(* PLC project WMT, Росатом LocalPLC 1, author Коробейников Петр *)
(* stored: creationDateTime 2021-03-09T09:02:31, contentDescription Система предиктивной диагностики. Модель теплового режима., productRelease 1, modificationDateTime 2023-03-16T09:01:23, language ru-RU, version 1, organization Филиал ВНИИЭФ НИИИС *)

TYPE P_INT : STRUCT
  A : INT := -1;
  B : INT := -1;
END_STRUCT;
END_TYPE

TYPE P_UINT : STRUCT
  A : UINT := 0;
  B : UINT := 0;
END_STRUCT;
END_TYPE

TYPE P_SINT : STRUCT
  A : SINT;
  B : SINT;
END_STRUCT;
END_TYPE

TYPE P_IDPIT : STRUCT
  A : UINT := 0;
  B : TPos8 := -1;
END_STRUCT;
END_TYPE

TYPE P_SIBT : STRUCT
  A : SINT := 0;
  B : BYTE := 0;
END_STRUCT;
END_TYPE

TYPE P_BOOL : STRUCT
  A : BOOL := false;
  B : BOOL := false;
END_STRUCT;
END_TYPE

TYPE TDef : STRUCT
  ID : UINT := 0;
  CF : WORD := 0;
  R0 : INT := 0;
  XYZ : ARRAY[0..2] OF INT := [0, 0, 0];
  LWH : ARRAY[0..2] OF INT := [100, 100, 100];
  Ig : SINT := 0;
  Im : SINT := 0;
  Iv : SINT := 0;
END_STRUCT;
END_TYPE

TYPE TMat : STRUCT
  KT : REAL := 0.11;
  CP : REAL := 1666.0;
  PL : REAL := 880.3;
  MD : REAL := 198.1;
END_STRUCT;
END_TYPE

TYPE TRad : STRUCT
  Vm : REAL := 0.02;
  Fk : REAL := 1.1;
  Q0 : REAL := 0.003;
  Q1 : REAL := 0.01;
  BL : ARRAY[0..3] OF REAL := [0.2, 0.6, 0.85, 1.0];
END_STRUCT;
END_TYPE

TYPE THead : STRUCT
  Ni : SINT := 0;
  Ng : SINT := 0;
  Nm : SINT := 0;
  Nv : SINT := 0;
  Np : SINT := 0;
  Ri : SINT := 0;
  ID : UINT := 0;
  TR : ARRAY[0..3] OF TIME := [T#60s, T#30s, T#10s, T#5s];
  Ax : UINT := 0;
  pX : INT := 0;
  pY : INT := 0;
  pZ : INT := 0;
  RV : ARRAY[0..1] OF DINT := [0, 0];
END_STRUCT;
END_TYPE

TYPE TRes : STRUCT
  DR : UDINT := 0;
  TR : TIME := T#0s;
  FP : TIME := T#0s;
  ER : UINT := 0;
  FL : WORD := 0;
  RV : ARRAY[0..5] OF UDINT := [0, 0, 0, 0, 0, 0];
END_STRUCT;
END_TYPE

TYPE TVal : STRUCT
  Iv : INT := 0;
  Vi : ARRAY[0..2] OF P_SINT := [0, 0, 0];
END_STRUCT;
END_TYPE

TYPE TProf : ARRAY[0..11] OF P_SINT;
END_TYPE

TYPE TConf : STRUCT
  Nm : UINT := 0;
  Nr : UINT := 0;
  Tc : TIME := T#10s;
END_STRUCT;
END_TYPE

TYPE TPhaseI : STRUCT
  Ic : REAL := 100.0;
  Tin : REAL := 40.0;
  Tout : REAL := 80.0;
  Rn : DWORD := 16#FFFF;
  RD : ARRAY[0..7] OF P_SINT := [0, 0, 0, 0, 0, 0, 0, 0];
END_STRUCT;
END_TYPE

TYPE TPhaseO : STRUCT
  Q0 : REAL := 0.0;
  Q1 : REAL := 0.0;
  Q2 : REAL := 0.0;
  Tin : REAL := 20.0;
  Tout : REAL := 80.0;
  Qm : REAL := 0.01;
  Se : REAL := 0.01;
  Ve : REAL := 0.01;
END_STRUCT;
END_TYPE

TYPE TCond : STRUCT
  ID : UINT := 0;
  Tmid : INT := 0;
  Tmin : TDot;
  Tmax : TDot;
END_STRUCT;
END_TYPE

TYPE TVarI : STRUCT
  DTI : UDINT := 0;
  TMI : TIME := T#0s;
  TOV : REAL := 0.0;
  MHT : REAL := 0.0;
  RI1 : REAL := 0.0;
  RI2 : REAL := 0.0;
END_STRUCT;
END_TYPE

TYPE TVarO : STRUCT
  DTO : UDINT := 0;
  TMO : TIME := T#0s;
  QTY : REAL := 0.0;
  QTS : REAL := 0.0;
  RO1 : REAL := 0.0;
  RO2 : REAL := 0.0;
END_STRUCT;
END_TYPE

TYPE TError : (E_SUCCESS, E_ID, E_HEAD, E_INDEX, E_ITEMPOS, E_ITEM, E_GRID, E_AXIS, E_PRIO, E_MATER, E_PROFILE, E_VALUE, E_STACKSIZE, E_ROOT, E_ITEMSIZE, E_STEPSIZE, E_TIMESIZE, E_NOTREADY, E_STRUCT, E_VALIDATE, E_LOC2ABS, E_ABS2LOC, E_GETTEMP, E_SETTEMP, E_CHECKVALID, E_LINKITEMS, E_PROCESS, E_PREPROC, E_POSTPROC, E_BADTEMP, E_STATE, E_CHECK, E_FAIL, W_PERIOD) := E_SUCCESS;
END_TYPE

TYPE TDir : (DIR_UP, DIR_DOWN);
END_TYPE

TYPE TIter : STRUCT
  dir : TDir := DIR_UP;
  prev : TPos8 := -1;
  item : TPos8 := -1;
  next : TPos8 := -1;
  last : TPos8 := -1;
  stack : ARRAY[0..3] OF TPos8 := [0, 0, 0, 0];
END_STRUCT;
END_TYPE

TYPE TPoint : ARRAY[0..2] OF REAL;
END_TYPE

TYPE TAxO : STRUCT
  x : USINT := 0;
  y : USINT := 0;
  z : USINT := 0;
END_STRUCT;
END_TYPE

TYPE P_RESI : STRUCT
  A : REAL := 0.0;
  B : SINT := 0;
END_STRUCT;
END_TYPE

TYPE P_RERE : STRUCT
  A : REAL := 0.0;
  B : REAL := 0.0;
END_STRUCT;
END_TYPE

TYPE TMatter : STRUCT
  a : REAL := 0.0001;
  l : REAL := 1.0;
  h : REAL := 0.001;
  k : REAL := 1.0;
END_STRUCT;
END_TYPE

TYPE TProps : STRUCT
  Air : BOOL := false;
  Oil : BOOL := false;
  Fluid : BOOL := false;
  Solid : BOOL := false;
END_STRUCT;
END_TYPE

TYPE LOGLEVEL : (CRITICAL, WARNING, INFO, DEBUG) := DEBUG;
END_TYPE

TYPE TStat : STRUCT
  RDY : BOOL := FALSE;
  DBG : BOOL := TRUE;
  ERR : TError := E_SUCCESS;
  PAR : UINT := 0;
  STR : STRING := '';
END_STRUCT;
END_TYPE

TYPE TGrid : STRUCT
  A : ARRAY[0..6271] OF TVar;
END_STRUCT;
END_TYPE

TYPE TVar : DINT;
END_TYPE

TYPE TDot : STRUCT
  V : INT := 0;
  A : TKnot := [0, 0, 0];
END_STRUCT;
END_TYPE

TYPE TShape : STRUCT
  wF : WORD := 0;
  Kn : TKnot := [0, 0, 0];
  p0 : TPoint := [0.0, 0.0, 0.0];
  pL : TPoint := [0.0, 0.0, 0.0];
  Lx : TPoint := [0.0, 0.0, 0.0];
END_STRUCT;
END_TYPE

TYPE TKnot : ARRAY[0..2] OF INT := [0, 0, 0];
END_TYPE

TYPE TItem : STRUCT
  ID : UINT := 0;
  Im : SINT := -1;
  Iv : SINT := -1;
  PDT : ARRAY[0..2] OF DT := [t#0ms, t#0ms, t#0ms];
  Par : TPos8 := -1;
  Num : SINT := 0;
  Kids : ARRAY[0..15] OF TPos8 := [0, 0, 0, 0, 0, 0, 0, 0, 0, 0, 0, 0, 0, 0, 0, 0];
END_STRUCT;
END_TYPE

TYPE TPos16 : INT := -1;
END_TYPE

TYPE TPos8 : SINT := -1;
END_TYPE

TYPE TItems : STRUCT
  Pr : ARRAY[0..99] OF P_IDPIT := [0, 0, 0, 0, 0, 0, 0, 0, 0, 0, 0, 0, 0, 0, 0, 0, 0, 0, 0, 0, 0, 0, 0, 0, 0, 0, 0, 0, 0, 0, 0, 0, 0, 0, 0, 0, 0, 0, 0, 0, 0, 0, 0, 0, 0, 0, 0, 0, 0, 0, 0, 0, 0, 0, 0, 0, 0, 0, 0, 0, 0, 0, 0, 0, 0, 0, 0, 0, 0, 0, 0, 0, 0, 0, 0, 0, 0, 0, 0, 0, 0, 0, 0, 0, 0, 0, 0, 0, 0, 0, 0, 0, 0, 0, 0, 0, 0, 0, 0, 0];
  It : ARRAY[0..99] OF TItem := [0, 0, 0, 0, 0, 0, 0, 0, 0, 0, 0, 0, 0, 0, 0, 0, 0, 0, 0, 0, 0, 0, 0, 0, 0, 0, 0, 0, 0, 0, 0, 0, 0, 0, 0, 0, 0, 0, 0, 0, 0, 0, 0, 0, 0, 0, 0, 0, 0, 0, 0, 0, 0, 0, 0, 0, 0, 0, 0, 0, 0, 0, 0, 0, 0, 0, 0, 0, 0, 0, 0, 0, 0, 0, 0, 0, 0, 0, 0, 0, 0, 0, 0, 0, 0, 0, 0, 0, 0, 0, 0, 0, 0, 0, 0, 0, 0, 0, 0, 0];
  Sh : ARRAY[0..100] OF TShape := [0, 0, 0, 0, 0, 0, 0, 0, 0, 0, 0, 0, 0, 0, 0, 0, 0, 0, 0, 0, 0, 0, 0, 0, 0, 0, 0, 0, 0, 0, 0, 0, 0, 0, 0, 0, 0, 0, 0, 0, 0, 0, 0, 0, 0, 0, 0, 0, 0, 0, 0, 0, 0, 0, 0, 0, 0, 0, 0, 0, 0, 0, 0, 0, 0, 0, 0, 0, 0, 0, 0, 0, 0, 0, 0, 0, 0, 0, 0, 0, 0, 0, 0, 0, 0, 0, 0, 0, 0, 0, 0, 0, 0, 0, 0, 0, 0, 0, 0, 0, 0];
  Cn : ARRAY[0..100] OF TCond := [0, 0, 0, 0, 0, 0, 0, 0, 0, 0, 0, 0, 0, 0, 0, 0, 0, 0, 0, 0, 0, 0, 0, 0, 0, 0, 0, 0, 0, 0, 0, 0, 0, 0, 0, 0, 0, 0, 0, 0, 0, 0, 0, 0, 0, 0, 0, 0, 0, 0, 0, 0, 0, 0, 0, 0, 0, 0, 0, 0, 0, 0, 0, 0, 0, 0, 0, 0, 0, 0, 0, 0, 0, 0, 0, 0, 0, 0, 0, 0, 0, 0, 0, 0, 0, 0, 0, 0, 0, 0, 0, 0, 0, 0, 0, 0, 0, 0, 0, 0, 0];
  Gr : ARRAY[0..99] OF TGrid := [0, 0, 0, 0, 0, 0, 0, 0, 0, 0, 0, 0, 0, 0, 0, 0, 0, 0, 0, 0, 0, 0, 0, 0, 0, 0, 0, 0, 0, 0, 0, 0, 0, 0, 0, 0, 0, 0, 0, 0, 0, 0, 0, 0, 0, 0, 0, 0, 0, 0, 0, 0, 0, 0, 0, 0, 0, 0, 0, 0, 0, 0, 0, 0, 0, 0, 0, 0, 0, 0, 0, 0, 0, 0, 0, 0, 0, 0, 0, 0, 0, 0, 0, 0, 0, 0, 0, 0, 0, 0, 0, 0, 0, 0, 0, 0, 0, 0, 0, 0];
  Gr2 : ARRAY[0..1] OF TGrid2 := [0, 0];
END_STRUCT;
END_TYPE

TYPE TSets : STRUCT
  Mt : ARRAY[0..11] OF TMat := [0, 0, 0, 0, 0, 0, 0, 0, 0, 0, 0, 0];
  Vl : ARRAY[0..24] OF TVal := [0, 0, 0, 0, 0, 0, 0, 0, 0, 0, 0, 0, 0, 0, 0, 0, 0, 0, 0, 0, 0, 0, 0, 0, 0];
  Pr : ARRAY[0..29] OF TProf := [0, 0, 0, 0, 0, 0, 0, 0, 0, 0, 0, 0, 0, 0, 0, 0, 0, 0, 0, 0, 0, 0, 0, 0, 0, 0, 0, 0, 0, 0];
  Bf : ARRAY[0..31] OF REAL := [0, 0, 0, 0, 0, 0, 0, 0, 0, 0, 0, 0, 0, 0, 0, 0, 0, 0, 0, 0, 0, 0, 0, 0, 0, 0, 0, 0, 0, 0, 0, 0];
END_STRUCT;
END_TYPE

TYPE THandle : ULINT;
END_TYPE

TYPE TGrid2 : STRUCT
  A : ARRAY[0..12543] OF TVar;
END_STRUCT;
END_TYPE

(* Дескриптор массива ITS.GR *)
FUNCTION its_gr2 : THandle
  VAR_INPUT
    Off : TPos8 := 0;  (* Опорная позиция сетки *)
  END_VAR

            {{ ITS_GR2 = (THANDLE)&__GET_GLOBAL_ITS()->GR2.table[OFF]; }}

          
END_FUNCTION

(* Дескриптор массива ITS.GR *)
FUNCTION its_gr : THandle
  VAR_INPUT
    Off : TPos8 := 0;  (* Опорная позиция сетки *)
  END_VAR

            {{ ITS_GR = (THANDLE)&__GET_GLOBAL_ITS()->GR.table[OFF]; }}

          
END_FUNCTION

(* Возвращает фигуру элемента *)
FUNCTION get_sh : TShape
  VAR_INPUT
    PSH : TPos8 := -1;  (* Позиция фигуры элемента *)
  END_VAR

            {{ return (GET_SH = __GET_GLOBAL_ITS()->SH.table[PSH]); }}

          
END_FUNCTION

(* Поиск в массиве IDS по ID *)
FUNCTION ID2PIT : TPos8
  VAR_INPUT
    ID : UINT := 0;  (* Идентификатор элемента *)
  END_VAR
  VAR
    bFound : BOOL := false;  (* Флаг - элемент найден *)
  END_VAR

            {{
  ID2PIT = -1;
  P_IDPIT *IDS = &(__GET_GLOBAL_ITS()->PR.table[0]);
  if (ID != 0) {
    int lBound=0, rBound=99, test;
    if (IDS[rBound].A == ID)      ID2PIT = IDS[rBound].B;
    else if (IDS[lBound].A == ID) ID2PIT = IDS[lBound].B;
    else {
      if ( (IDS[lBound].A < ID) && (ID < IDS[rBound].A) ) {
        while (TRUE) {
          test = (lBound+rBound)/2;
          if (IDS[test].A == ID) { ID2PIT = IDS[test].B; break; }
          if (rBound-lBound <= 1) break;
          if (IDS[test].A <  ID) lBound = test; else rBound = test; 
        }
      }
    }
  } else ID2PIT = IDS[0].B;
}}
          
END_FUNCTION

(* TRUE, если элемент - родитель *)
FUNCTION is_poly : BOOL
  VAR_INPUT
    PIT : TPos8 := -1;  (* Позиция элемента *)
  END_VAR

            {{ 
  return (IS_POLY = (__GET_GLOBAL_ITS()->IT.table[PIT].NUM > 0)); 
}}

          
END_FUNCTION

(* Терминальный итератор *)
FUNCTION it_end : TIter
  VAR_INPUT
    PIT : TPos8 := -1;  (* Признак терминального узла *)
  END_VAR

            {{ 
  return (IT_END = ((TITER){ TDIR__DIR_UP, -1, -1, -1, -1, {0,0,0,0} } )); 
}}

          
END_FUNCTION

(* Аварийное завершение программы *)
FUNCTION halt : BOOL
  VAR_INPUT
    ERR : TError := E_FAIL;  (* Код ошибки *)
  END_VAR

            (* Использует вызов sleep() и exit() для завершения потоков *)
{{
  //#ifndef __ASSERT_H
  //#define __ASSERT_H 1
     //#include <unistd.h> // Include "unistd.h" for sleep() & exit() function
  //#endif // __ASSERT_H
  //sleep(3); // Wait for message logging..
  //exit(ERR);
}}
          
END_FUNCTION

(* Приоритет по коду ошибки *)
FUNCTION Err2Lev : LOGLEVEL
  VAR_INPUT
    Err : TError := E_SUCCESS;  (* Флаг ошибки *)
  END_VAR

            CASE Err OF
E_SUCCESS:  
  Err2Lev:=INFO;  
W_PERIOD:   
  Err2Lev:=WARNING;  
ELSE        
  Err2Lev:=CRITICAL;  
END_CASE;
RETURN;
          
END_FUNCTION

(* Выдает строку по коду ошибки *)
FUNCTION Err2Str : STRING
  VAR_INPUT
    ERR : TError := E_SUCCESS;  (* Код ошибки *)
  END_VAR

            case ERR of
(* Информационные сообщения *)
E_SUCCESS:      Err2Str := 'Succeeded!';

(* Критические ошибки *)
E_FAIL:         Err2Str := 'Unexpected error';
E_STATE:        Err2Str := 'Program state error';
E_CHECK:        Err2Str := 'Check point error';
E_HEAD:         Err2Str := 'Invalid head';
E_INDEX:        Err2Str := 'Invalid index';
E_ITEMPOS:      Err2Str := 'Invalid item position';
E_ITEM:         Err2Str := 'Invalid element';
E_GRID:         Err2Str := 'Invalid grid';
E_AXIS:         Err2Str := 'Invalid axis';
E_PRIO:         Err2Str := 'Invalid prio';
E_MATER:        Err2Str := 'Invalid mater';
E_PROFILE:      Err2Str := 'Invalid profile';
E_VALUE:        Err2Str := 'Invalid value';
E_ROOT:         Err2Str := 'Invalid ROOT';
E_ITEMSIZE:     Err2Str := 'Bad ItemAt size';
E_STEPSIZE:     Err2Str := 'Bad axis step';
E_TIMESIZE:     Err2Str := 'Bad time step';
E_STACKSIZE:    Err2Str := 'Small stacksize';
E_NOTREADY:     Err2Str := 'Object dont ready';
E_LOC2ABS:      Err2Str := 'Loc2Abs error';
E_ABS2LOC:      Err2Str := 'Abs2Loc error';
E_VALIDATE:     Err2Str := 'Validate error';
E_CHECKVALID:   Err2Str := 'CheckValid error';
E_LINKITEMS:    Err2Str := 'LinkItems error';
E_PROCESS:      Err2Str := 'Process item error';
E_BADTEMP:      Err2Str := 'GetTemp error';

(* Предупреждения *)
W_PERIOD:       Err2Str := 'Small period';
else            Err2Str := 'Unknown error';
end_case;

          
END_FUNCTION

(* Протоколирование ошибки *)
FUNCTION LogMsg : STRING
  VAR_INPUT
    STR : STRING := '';  (* Строка для протокола *)
    LVL : LOGLEVEL := DEBUG;  (* Уровень сообщения (по умолчанию - Debug) *)
    ERR : TError := E_SUCCESS;  (* Код ошибки *)
  END_VAR

            {{
  #ifdef _BEREMIZ_H_
    #define __LOG_MSG(level,string,length) LogMessage(level,(char *)string,length)
  #else
    #define __LOG_MSG(level,string,length) printf("%s\n", (char *)string)
  #endif
  TSTAT *pStat = __GET_GLOBAL_STAT();
  if (LVL!=LOGLEVEL__DEBUG || (LVL==LOGLEVEL__DEBUG && pStat->DBG)) {
    if (STR.len) __LOG_MSG(LVL, (char *)STR.body, STR.len);
  }
  if (ERR!=TERROR__E_SUCCESS) {
    pStat->ERR=ERR;
    LVL=ERR2LEV(1,NULL,ERR); 
    STR=ERR2STR(1,NULL,ERR);
    if (STR.len) __LOG_MSG(LVL,(char *)STR.body,STR.len);
  }
  return (LOGMSG = __INIT_STRING);
}}

          
END_FUNCTION

(* Выдает строку по коду ошибки *)
FUNCTION MakeMsg : STRING
  VAR_INPUT
    S0 : STRING := '';  (* Строка 0 *)
    S1 : STRING := '';  (* Строка 1 *)
    S2 : STRING := '';  (* Строка 2 *)
    S3 : STRING := '';  (* Строка 3 *)
  END_VAR
  VAR
    BLOG : BOOL := FALSE;  (* Флаг работы *)
  END_VAR

            {{ BLOG = __GET_GLOBAL_STAT()->DBG; }}
if (BLOG) then 
  MakeMsg:=concat(concat(concat(S0, S1), S2), S3); 
else 
  MakeMsg:=''; 
end_if;
          
END_FUNCTION

(* Аналог функции assert в C *)
FUNCTION assert : BOOL
  VAR_INPUT
    STAT : BOOL := FALSE;  (* Выражение для утверждения *)
    ERR : TError := E_FAIL;  (* Код ошибки *)
    STR : STRING := '';  (* Строка в лог *)
  END_VAR

            {{
//  #ifndef __ASSERT_H
//  #define __ASSERT_H 1
//     #include <unistd.h> // Include "unistd.h" for sleep() & exit() function
//     #include <assert.h> // Include "unistd.h" for sleep() & exit() function
//  #endif // __ASSERT_H
  if (!(ASSERT=STAT)) { 
    STR = MAKEMSG(1, NULL, 
      __STRING_LITERAL(27,"OpenPLC: ASSERTION FAILED! "), 
      STR,
      __INIT_STRING,
      __INIT_STRING
    );
    LOGMSG(1, NULL, STR, LOGLEVEL__CRITICAL, ERR); 
    //HALT(1, NULL, ERR);
    //sleep(3); // Wait for message logging..
    //exit(ERR);
//    assert(0);
  }
}}
          
END_FUNCTION

(* Уровень вложенности элемента *)
FUNCTION it_lev : SINT
  VAR_INPUT
    PIT : TPos8 := -1;
  END_VAR
  VAR
    IID : UINT := 16#ffff;
  END_VAR

            {{
  IID = __GET_GLOBAL_ITS()->IT.table[PIT].ID;
  if (IID==0 || IID==0xffff) return (IT_LEV=-1);
  IT_LEV = 3;
  if (IID & 0x000F) return(IT_LEV); IT_LEV--;
  if (IID & 0x00F0) return(IT_LEV); IT_LEV--;
  if (IID & 0x0F00) return(IT_LEV); IT_LEV--;
}}

          
END_FUNCTION

(* Обход дерева элементов *)
FUNCTION it_next : TIter
  VAR_INPUT
    it : TIter;  (* Итератор *)
  END_VAR

            {{ 
  /* Алгоритм обхода:
    1) Если предыдущий узел - родительский для этого узла 
       -> переходим к первому дочернему узлу (если нет->к родителю);
    2) Если предыдущий узел - дочерний для этого узла  
       -> переходим к следующему дочернему узлу (если нет->к родителю) 
  */
  SINT iSub = 0;
  SINT iLevel = 0;
  BOOL bBreak = FALSE;
  TITEM *Items = &(__GET_GLOBAL_ITS()->IT.table[0]);
  
  while (!bBreak && IT.ITEM!=(-1)) { 
    IT.ITEM = IT.NEXT;  // Переход к следующему элементу
    if (IT.ITEM!=(-1)) {
      // Запоминаем уровень текущего узла в стеке со смещением +1
      iLevel = IT_LEV(1,NULL,IT.ITEM)+1; 
      
      // Определение следующего узла
      if (IT.PREV == Items[IT.ITEM].PAR) {
        // предыдущий узел является является родительским узлом этого узла ->
        iSub = 0;
        if (Items[IT.ITEM].NUM > iSub) { 
          // ВНИЗ -> к первому дочернему узлу (если есть)
          IT.NEXT = Items[IT.ITEM].KIDS.table[iSub];
          IT.STACK.table[iLevel] = iSub;
          IT.DIR = TDIR__DIR_DOWN;  // Актуально если есть потомки
          bBreak = TRUE; 
        } else {    
          // ВВЕРХ -> к родителю (потомков нет)
          IT.NEXT = (IT.ITEM != IT.LAST) ? IT.NEXT = Items[IT.ITEM].PAR : (-1);
          IT.DIR = TDIR__DIR_UP;    // Актуально для любого элемента
          bBreak = TRUE;
        }
      } else if (Items[IT.PREV].PAR == IT.ITEM) { 
        // предыдущий узел является дочерним узлом этого узла ->
        iSub = IT.STACK.table[iLevel]+1;
        if (iSub < Items[IT.ITEM].NUM) {
          // ПО ГОРИЗОНТАЛИ -> к следующему дочернему узлу (если есть)
          IT.NEXT = Items[IT.ITEM].KIDS.table[iSub];
          IT.STACK.table[iLevel] = iSub;
        } else {
          // ВВЕРХ -> к родителю (потомков больше нет)
          IT.NEXT = (IT.ITEM != IT.LAST) ? IT.NEXT = Items[IT.ITEM].PAR : (-1);
          IT.DIR = TDIR__DIR_UP;
          bBreak = TRUE;
        }
      } else {
        //ASSERT(1,NULL,FALSE, TERROR__E_FAIL, 
          //__STRING_LITERAL(24,"it_next: Bad struct!"));
        return (IT_NEXT = IT_END(1,NULL,-1)); // так не бывает - ошибка структуры!!!
      }
    }
    IT.PREV = IT.ITEM;  // Сохранение текущего узла
  }
  return (IT_NEXT = IT);
}}

          
END_FUNCTION

(* Итератор дерева элементов *)
FUNCTION it_begin : TIter
  VAR_INPUT
    PIT : TPos8 := -1;  (* Начальный индекс элемента *)
  END_VAR
  VAR
    bValid : BOOL := true;  (* Флаг валидности начальной позиции *)
  END_VAR

            (* Инициализация итератора *)
{{
  BOOL bValid = (PIT >= 0 && PIT < __GET_GLOBAL_HDR()->NI);
  if (bValid) {
    IT_BEGIN.PREV = __GET_GLOBAL_ITS()->IT.table[PIT].PAR;
    IT_BEGIN.ITEM = IT_BEGIN.NEXT = IT_BEGIN.LAST = PIT;
    // Если позиция начала верна - делаем первую итерацию
    return (IT_BEGIN = IT_NEXT(1,NULL,IT_BEGIN));
  } else 
      // Если позиция не верна - переход в конечное состояние
      return (IT_BEGIN = IT_END(1,NULL,(-1)));
}}

          
END_FUNCTION

(* Нормирование диапазона угла *)
FUNCTION angle : REAL
  VAR_INPUT
    A : REAL := 0.0;  (* Угол или угловой размер в градусах *)
    L0 : REAL := 0.0;  (* Начало отсчёта (по умолчанию = 0) *)
    PI2 : REAL := 360.0;  (* Диапазон (по умолчанию = 2*Пи в градусах) *)
  END_VAR

            (* Приведение аргумента к диапазону [L0..L0+2*PI] *)
while (A < L0    ) do A := A+PI2; end_while;
while (A > L0+PI2) do A := A-PI2; end_while;
angle := A;
          
END_FUNCTION

(* Порядок координатных осей x,y,z *)
FUNCTION AxO : TAxO
  VAR_INPUT
    Ax : USINT := 0;  (* Ориентация оси симметрии *)
    inside : BOOL := TRUE;  (* Флаг преобразования "Изнутри" *)
  END_VAR

            (*  Порядок координат при различной ориентации оси *)
if (inside) then
  (* Взгляд изнутри: какой индекс в локальных координатах элемента
    X(R),Y(F),Z имеет абсолютная координата (Ox,Oy,Oz)
    при заданной ориентации оси симметрии Ax?
  (* Индексы координат, ставших X,Y,Z:  Ax  | 1 | 2 | 3 | *)
  (* O.x-индекс радиуса,O.y-угол,O.z-высота ------------- *)
  AxO.x := (0+Ax) mod 3; (* Ind_of_X  (O.x) | 1 | 2 | 0 | *)
  AxO.y := (1+Ax) mod 3; (* Ind_of_Y  (O.y) | 2 | 0 | 1 | *)  
  AxO.z := (2+Ax) mod 3; (* Ind_of_Z  (O.z) | 0 | 1 | 2 | *)
else  (* Обратное преобразование -> *)
  (* Взгляд снаружи: какую роль абсолютная координата (Ox,Oy,Oz)
     играет для вложенного во внешнюю систему элемента?   *)
  (* Порядок "перебора" координат:  Ax=Ix+1 | 1 | 2 | 3 | *)
  (* где 0-внешний цикл, 2-самый вложенный  ------------- *)
  AxO.x := (3-Ax) mod 3; (* Ind_of_X  (O.x) | 2 | 1 | 0 | *)
  AxO.y := (4-Ax) mod 3; (* Ind_of_Y  (O.y) | 0 | 2 | 1 | *)  
  AxO.z := (5-Ax) mod 3; (* Ind_of_Z  (O.z) | 1 | 0 | 2 | *)
end_if;
          
END_FUNCTION

(* Генератор импульсов по времени *)
FUNCTION_BLOCK FRONT
  VAR_INPUT
    IN : BOOL := TRUE;  (* Деблокировка блока *)
    PT : TIME := T#1s;  (* Период отсчета таймера *)
  END_VAR
  VAR_OUTPUT
    OUT : BOOL := FALSE;  (* Передний фронт (держится 1 цикл) *)
    INV : BOOL := FALSE;  (* Инверсия переднего фронта *)
  END_VAR
  VAR
    f_TP : TP := IN := FALSE;  (* Таймер задежки фронта TP *)
    f_TP_ET : TIME := T#0s;  (* Счетчик времени (0..TP) *)
    f_TP_Q : BOOL := FALSE;  (* Выход таймера TP *)
  END_VAR

            VAR
  (*Run    : R_TRIG;*)
  bReStart : BOOL   := TRUE;
END_VAR
  
(*Run(CLK := IN);*)
IF (IN) THEN
  IF ((*Run.Q*)bReStart) THEN     
    bReStart := FALSE;
    (* Инициализация *)
    f_TP(IN := FALSE);
    f_TP(IN := TRUE, PT := PT, Q => f_TP_Q, ET => f_TP_ET);
    OUT := TRUE;      (* Взвод триггера *)
  END_IF; 
  (* Нормальная работа *)
  (* Отсчет таймера *)
  f_TP(IN := FALSE, PT := PT, Q => f_TP_Q, ET => f_TP_ET);
  
  (* Анализ результата *)
  IF (f_TP.Q = FALSE) THEN 
    (* если отсчет закончился и ... *)
    IF (OUT = FALSE) THEN 
      (* ... если выход сброшен, тогда сразу начинаем новый отсчет *)
      f_TP(IN := TRUE, PT := PT, Q => f_TP_Q, ET => f_TP_ET);
      OUT := TRUE;  (* Взвод триггера *)
    ELSE 
      (* ... если выход взведен, то один цикл нужно пропустить !!! *)
      OUT := FALSE; (* Сброс триггера *)
    END_IF;
  ELSE
    OUT := FALSE;   (* Сброс триггера *)
  END_IF;
ELSE
  bReStart := TRUE;
END_IF; (* IN *)

(* Устанавливаем инверсный выход *)
IF (OUT <> TRUE) THEN INV := TRUE; ELSE INV := FALSE; END_IF;
  
RETURN;
          
END_FUNCTION_BLOCK

(* Градусы в радианы *)
FUNCTION radi : REAL
  VAR_INPUT
    GRA : REAL := 0.0;  (* Градусы *)
  END_VAR

            radi:=GRA*0.01745329251994329576923690768489;
          
END_FUNCTION

(* Расчёт деформации элемента *)
FUNCTION Reform : TPoint
  VAR_INPUT
    wF : WORD := 0;  (* Флаги границ элемента *)
    Ang : REAL := 0.0;  (* Угол развертки *)
    Pt : REAL := 0.0;  (* Локальная координата точки *)
    pL : REAL := 0.0;  (* Начальная координата точка *)
    Lx : REAL := 0.0;  (* Размер по координате *)
  END_VAR
  VAR
    pR : REAL := 0.0;  (* Конечная координата точки *)
    LR : P_BOOL;  (* Флаги формы границ *)
    Q : SINT := 0;  (* Индекс квадранта *)
    K : REAL := 0.0;  (* Коэффициент пропорциональности *)
    Kx : REAL := 0.0;  (* Коэффициент коррекции *)
  END_VAR
  VAR CONSTANT
    PI_2 : REAL := 90.0;  (* Число Пи/2 *)
    PI_4 : REAL := 45.0;  (* Число Пи/4 *)
    PI : REAL := 180.0;  (* Число Пи/2 *)
    PI3_2 : REAL := 270.0;  (* Число 3*Пи/2 *)
  END_VAR

            (* Нормируем угол 0-360 град. *)
Ang:=angle(Ang);

(* Определяем номер квадранта Q = [0..3] *)
if (Ang >= 0.0) then
  if    (Ang >= 0.0   and Ang <  PI_2 ) then Q := 0; 
  elsif (Ang >= PI_2  and Ang <  PI   ) then Q := 1; 
  elsif (Ang >= PI    and Ang <  PI3_2) then Q := 2; 
  else Q := 3;
  end_if;
else
  if    (Ang <= 0.0   and Ang > -PI_2 ) then Q := 3; 
  elsif (Ang <= -PI_2 and Ang > -PI   ) then Q := 2; 
  elsif (Ang <= -PI   and Ang > -PI3_2) then Q := 1; 
  else Q := 0;
  end_if;
end_if;

(* Определяем форму границ в квадранте Q *)
LR.A := ((wF and shl(16#10, Q))<>0);
LR.B := ((wF and shl(16#01, Q))<>0);

(* Делаем преобразование границ и точки Pt *)
if (LR.A or LR.B) then 
  (* Растяжение по радиусу от угла *)
  Ang := angle(Ang, 0.0, PI_2); 
  if (Ang < PI_4) 
  then Kx := 1.0/cos(radi(Ang));    (* коэффициент растяжения         *)
  else Kx := 1.0/sin(radi(Ang));    (* коэффициент растяжения         *)
  end_if;
  pR := pL + Lx;                    (* координата правой границы      *)
  K  := (Pt - pL)/Lx;               (* коэффициент пропорциональности *)
  if (LR.A) then pL:=pL*Kx; end_if; (* коррекция левой  границы       *)
  if (LR.B) then pR:=pR*Kx; end_if; (* коррекция правой границы       *)
  Lx := (pR - pL);                  (* размер по координате           *)
  Pt := pL + K * Lx;                (* координата точки               *)
end_if;

Reform[0] := Pt; (* текущая   координата *)
Reform[1] := pL; (* начальная координата *)
Reform[2] := Lx; (* размер по координате *)
          
END_FUNCTION

(* Радианы в градусы *)
FUNCTION grad : REAL
  VAR_INPUT
    RAD : REAL := 0.0;  (* Радианы *)
  END_VAR

            grad:=RAD*57.295779513082320876798154814105;
          
END_FUNCTION

(* Направление оси симметрии *)
FUNCTION sh_get_ax : USINT
  VAR_INPUT
    SH : TShape;  (* Фигура элемента *)
  END_VAR

            sh_get_ax := WORD_TO_USINT(SHR((Sh.wF AND 16#3000), 12));
          
END_FUNCTION

(* Сборка точки *)
FUNCTION _point : TPoint
  VAR_INPUT
    X : REAL := 0.0;  (* Координата X *)
    Y : REAL := 0.0;  (* Координата Y *)
    Z : REAL := 0.0;  (* Координата Z *)
  END_VAR

            {{ 
  _POINT.table[0] = X; 
  _POINT.table[1] = Y; 
  _POINT.table[2] = Z; 
}}

          
END_FUNCTION

(* Абс->Лок координаты *)
FUNCTION Sh_Abs2Loc : TPoint
  VAR_INPUT
    Sh : TShape;  (* Фигура элемента *)
    X : REAL := 0.0;  (* Точка, координата X (abs, декарт) *)
    Y : REAL := 0.0;  (* Точка, координата Y (abs, декарт) *)
    Z : REAL := 0.0;  (* Точка, координата Z (abs, декарт) *)
  END_VAR
  VAR
    Ax : USINT := 0;  (* Направление оси *)
    A : TPoint := [0.0, 0.0, 0.0];  (* Точка в координатах элемента *)
    B : TPoint := [0.0, 0.0, 0.0];  (* Вспомогательная точка *)
    O : TAxO;  (* Индексы координат x, y, z *)
    PI : REAL := 3.1415926535897932384626433832795;  (* Число Пи *)
    PI_2 : REAL := 1.5707963267948966192313216916398;  (* Число Пи/2 *)
  END_VAR
  VAR CONSTANT
    RAD : BOOL := FALSE;  (* Признак радиан (по умолчанию в градусах) *)
    DX : REAL := 1.0E-5;  (* Допустимая погрешность *)
  END_VAR

            (* Sh := get_sh(PIT); *)
Ax := sh_get_ax(Sh);

A := _point(X-Sh.P0[0],Y-Sh.P0[1],Z-Sh.P0[2]); 
if (Ax > 0) then 
  (* Декарт -> Цилиндр *)
  O := AxO(Ax);
  B[O.x] := sqrt(A[O.x]*A[O.x] + A[O.y]*A[O.y]);
  if (abs(A[O.x]) < DX) then A[O.x] := 0.0; end_if;
  if (abs(A[O.y]) < DX) then A[O.y] := 0.0; end_if;
  (* интерпретация atan2(y,x) *)
  if (A[O.x] < 0.0) then 
    if (A[O.y] < 0.0) then  B[O.y] := atan(A[O.y]/A[O.x])-PI; 
    else                    B[O.y] := atan(A[O.y]/A[O.x])+PI; 
    end_if;
  else 
    if (A[O.x] > 0.0) then
      B[O.y] := atan(A[O.y]/A[O.x]);
    else (* A[O.x] = 0.0 *)
      if (A[O.y] < 0.0) then 
        B[O.y] := -PI_2;  
      else 
        if (A[O.y] > 0.0) then
          B[O.y] := PI_2;   
        else (* y = 0.0 *)
          B[O.y] := 0.0; 
        end_if;
      end_if;
    end_if;
  end_if;
  if (abs(B[O.y]) < DX) then B[O.y] := 0.0; end_if;
  if (not RAD) then B[O.y] := grad(B[O.y]); end_if;
  B[O.z] := A[O.z];
else 
  B := A;
end_if;
Sh_Abs2Loc := B; 

          
END_FUNCTION

(* Сборка координат узла *)
FUNCTION _knot : TKnot
  VAR_INPUT
    I : INT := 0;  (* Индекс X *)
    J : INT := 0;  (* Индекс Y *)
    K : INT := 0;  (* Индекс Z *)
  END_VAR

            _knot[0] := I; 
_knot[1] := J; 
_knot[2] := K; 

          
END_FUNCTION

(* Сборка координат узла *)
FUNCTION _dot : TDot
  VAR_INPUT
    V : INT := 0;  (* Значение *)
    i : INT := 0;  (* Индекс X *)
    j : INT := 0;  (* Индекс Y *)
    k : INT := 0;  (* Индекс Z *)
  END_VAR

            _dot.V := V; 
_dot.A := _knot(i,j,k); 

          
END_FUNCTION

(* Узел по координатам *)
FUNCTION Sh_Point2Dot : TDot
  VAR_INPUT
    Sh : TShape;  (* Фигура элемента *)
    X : REAL := 0.0;  (* Точка, координата X (abs, декарт) *)
    Y : REAL := 0.0;  (* Точка, координата Y (abs, декарт) *)
    Z : REAL := 0.0;  (* Точка, координата Z (abs, декарт) *)
    fChk : BOOL := TRUE;  (* Проверять принадлежность точки *)
  END_VAR
  VAR
    Hn : TPoint := [0.0, 0.0, 0.0];  (* Размерность сетки *)
    Ax : USINT := 0;  (* Направление оси *)
    pL : TPoint := [0.0, 0.0, 0.0];  (* Левая точка элемента (лок, декарт|цилиндр) *)
    pR : TPoint := [0.0, 0.0, 0.0];  (* Правая точка элемента (лок, декарт|цилиндр) *)
    pDL : TPoint := [0.0, 0.0, 0.0];  (* Левые границы с погрешностью *)
    pDR : TPoint := [0.0, 0.0, 0.0];  (* Правые границы с погрешностью *)
    Ox : TAxO;  (* Индексы координат x, y, z *)
    Pt : TPoint := [0.0, 0.0, 0.0];  (* Проверяемая точка (abs, декарт) *)
    Hx : TPoint := [0.0, 0.0, 0.0];  (* Шаг по сетке элемента (X,Y,Z) *)
    P : TPoint := [0.0, 0.0, 0.0];  (* Результат деформации *)
    B : BYTE := 0;  (* Результат проверки точки *)
    bRes : BOOL := true;  (* Булевый результат *)
  END_VAR
  VAR CONSTANT
    DX : REAL := 1.0E-5;  (* Допуск *)
  END_VAR

            Ax := sh_get_ax(Sh);

(* точка (X,Y,Z)->лок *)
Pt := Sh_Abs2Loc(Sh, X, Y, Z);

(* Коррекция границ при изменении формы *)
if (Ax<>0) then
  Ox := AxO(Ax);
  Pt[Ox.y]:=angle(Pt[Ox.y], Sh.pL[Ox.y]);
  P := Reform(Sh.wF, Pt[Ox.y], 0.0, Sh.pL[Ox.x], Sh.Lx[Ox.x]);
  Sh.pL[Ox.x] := P[1]; Sh.Lx[Ox.x] := P[2];
end_if;

if (fChk) then 
  (* B[0] - 0x01 (In)    - точка внутри элемента    *)
  (* B[1] - 0x02 (Left)  - точка на левой грани     *)
  (* B[2] - 0x04 (Right) - точка на правой грани    *)
  (* B[3] - 0x08 (Front) - точка на передней грани  *)
  (* B[4] - 0x10 (Back)  - точка на задней грани    *)
  (* B[5] - 0x20 (Down)  - точка на нижней грани    *)
  (* B[6] - 0x40 (Up)    - точка на верхней грани   *)
  (* B[7] - 0x80 (Err)   - ошибка (не используется) *)
  pL  := Sh.pL;
  pR  := _point(Sh.pL[0]+Sh.Lx[0], Sh.pL[1]+Sh.Lx[1], Sh.pL[2]+Sh.Lx[2]);
  
  pDL := _point((pL[0])*(1.0+DX), (pL[1])*(1.0+DX), (pL[2])*(1.0+DX));
  pDR := _point((pR[0])*(1.0-DX), (pR[1])*(1.0-DX), (pR[2])*(1.0-DX));
  
  (*
  pDL := _point( pL[0]+(Sh.Lx[0]*DX), pL[1]+(Sh.Lx[1]*DX), pL[2]+(Sh.Lx[2]*DX) );
  pDR := _point( pR[0]-(Sh.Lx[0]*DX), pR[1]-(Sh.Lx[1]*DX), pR[2]-(Sh.Lx[2]*DX) );
  *)
  
  (* Проверка: точка внутри элемента -> B=1 *)
  if ( (Pt[0] > pDL[0]) and (Pt[0] < pDR[0]) ) then 
    if ( (Pt[1] > pDL[1]) and (Pt[1] < pDR[1]) ) then
      if ( (Pt[2] > pDL[2]) and (Pt[2] < pDR[2]) ) then B:=16#01; end_if;
    end_if;
  end_if;
  
  (* Сравниваем координаты Pt с гранями элемента *)
  if (B = 0) then
    if    ( Pt[0] >= pL[0] and Pt[0] <= pDL[0] ) then B:=(B or shl(16#01, 1)); 
    elsif ( Pt[0] <= pR[0] and Pt[0] >= pDR[0] ) then B:=(B or shl(16#01, 2)); end_if;
    if    ( Pt[1] >= pL[1] and Pt[1] <= pDL[1] ) then B:=(B or shl(16#01, 3));
    elsif ( Pt[1] <= pR[1] and Pt[1] >= pDR[1] ) then B:=(B or shl(16#01, 4)); end_if;
    if    ( Pt[2] >= pL[2] and Pt[2] <= pDL[2] ) then B:=(B or shl(16#01, 5)); 
    elsif ( Pt[2] <= pR[2] and Pt[2] >= pDR[2] ) then B:=(B or shl(16#01, 6)); end_if;
  end_if;
  if (B = 0) then (* точка вне элемента *)
    {}(* bRes := assert(false, E_CHECK); *) 
  end_if;
end_if;

(* Получение узла сетки элемента *)
if (Sh.Kn[0]>1) then Hn[0]:=(Sh.Lx[0]/INT_TO_REAL(Sh.Kn[0]-1)); end_if;
if (Sh.Kn[1]>1) then Hn[1]:=(Sh.Lx[1]/INT_TO_REAL(Sh.Kn[1]-1)); end_if;
if (Sh.Kn[2]>1) then Hn[2]:=(Sh.Lx[2]/INT_TO_REAL(Sh.Kn[2]-1)); end_if;

Sh_Point2Dot := _dot(
    byte_to_int(B),
    min(Sh.Kn[0]-1, max(0, REAL_TO_INT((Pt[0]-Sh.pL[0])/Hn[0]) )), 
    min(Sh.Kn[1]-1, max(0, REAL_TO_INT((Pt[1]-Sh.pL[1])/Hn[1]) )), 
    min(Sh.Kn[2]-1, max(0, REAL_TO_INT((Pt[2]-Sh.pL[2])/Hn[2]) ))
);

          
END_FUNCTION

(* Проверка статуса ошибки *)
FUNCTION st_check : BOOL
  VAR_INPUT
    Force : BOOL := FALSE;  (* Флаг принудительного TRUE *)
  END_VAR

            {{ 
  return (
    ST_CHECK = ( 
      FORCE || (ERR2LEV(1,NULL,__GET_GLOBAL_STAT()->ERR) != LOGLEVEL__CRITICAL) 
    )
  ); 
}}

          
END_FUNCTION

(* Поиск владельцев точки (X,Y,Z) *)
FUNCTION Do_FindDot : TDot
  VAR_INPUT
    X : REAL := 0.0;  (* Координата X *)
    Y : REAL := 0.0;  (* Координата Y *)
    Z : REAL := 0.0;  (* Координата Z *)
    ign : TPos8 := -1;  (* Игнорируемый элемент *)
  END_VAR
  VAR
    It : TIter;  (* Итератор *)
    skip_to : TPos8 := -1;  (* Пропуск детей, если точка не у родителя *)
    i : SINT := 0;  (* Индекс перебора *)
    N : SINT := 0;  (* Количество найденных элементов *)
    Dots : ARRAY[0..7] OF TDot;  (* Массив найденных точек *)
    P : ARRAY[0..7] OF TPos8;  (* Найденные элементы *)
  END_VAR

            if (not st_check(false)) then return; end_if;

(* Обход дерева - сбор элементов, содержащих точку *)
it  := it_begin(ID2PIT(0));
while (it.item<>-1 and N < 8) do (* не более 8 владельцев *)
  case (it.dir) of
  DIR_DOWN:
    if (skip_to = -1) then
      (* Если точка не входит в родителя, потомков пропускаем *)
      if (is_poly(it.item)) then
        Do_FindDot := Sh_Point2Dot(get_sh(it.item), X, Y, Z);
        if (Do_FindDot.V <= 0) then skip_to := it.item; end_if;
      end_if;
    end_if;
  DIR_UP:
    if (skip_to <> -1) then
      if (skip_to = it.item) then skip_to := -1; end_if;
    else
      (* если элемент конечный - проверяем точку *)
      if (not is_poly(it.item)) then
        Dots[N] := Sh_Point2Dot(get_sh(it.item), X, Y, Z);
        if (Dots[N].V > 0) then 
          P[N] := it.item; 
          N    := N+1; 
        end_if;
      end_if;
    end_if;
  end_case;
  it := it_next(it);
end_while;

(* Выбор элемента *)
Do_FindDot := _dot(-1);
if (N > 0) then
  for i:=0 to N-1 do
  
    if (((*ign<>-1 and*) P[i]<>ign) or N=1) then 
        Do_FindDot   := Dots[i]; 
        Do_FindDot.V := sint_to_int(P[i]); 
       exit; 
    end_if;
    
  end_for;
end_if;
          
END_FUNCTION

(* Значение OFF типа P_INT *)
FUNCTION knoff : P_INT
  VAR_INPUT
    Nx : INT := 1;  (* Размер сетки по X *)
    Ny : INT := 1;  (* Размер сетки по Y *)
    Nz : INT := 1;  (* Размер сетки по Z *)
    I : INT := 0;  (* Индекс сетки-0 *)
    J : INT := 0;  (* Индекс сетки-1 *)
    K : INT := 0;  (* Индекс сетки-2 *)
  END_VAR

            knoff.A := 0;  (* начальное смещение 0-ячейки в массиве Grid *)
knoff.B := 1;  (* количество ячеек  в массиве Grid (min = 1) *)
if (K > 0) then
  knoff.A := knoff.A + K*2*(Nx+Ny) + (K+1)*Nx*Ny;
  if (K = (Nz-1)) then knoff.B := knoff.B+1; end_if;
else knoff.B := knoff.B+1;
end_if;
if (J > 0) then
  knoff.A := knoff.A + J*(2+knoff.B*Nx) + Nx;
  if (J = (Ny-1)) then knoff.B := knoff.B+1; end_if;
else knoff.B := knoff.B+1;
end_if;
if (I > 0) then
  knoff.A := knoff.A + I*knoff.B + 1;
  if (I = (Nx-1)) then knoff.B := knoff.B+1; end_if;
else knoff.B := knoff.B+1;
end_if;


          
END_FUNCTION

(* Задание значения типа TVar *)
FUNCTION set_var : TPos8
  VAR_INPUT
    HGR : THandle := 0;  (* Дескриптор массива сеток *)
    PGR : TPos8 := -1;  (* Позиция сетки в массиве *)
    OFF : P_INT;  (* Смещение узла в сетке *)
    TV : TVar := -1;  (* Значение ячейки узла сетки *)
    IX : USINT := 0;  (* Ключ направления (0xff-неопределён) *)
  END_VAR

            {{
  #pragma pack(push, 4)
  typedef union {
    TVAR tv;
    struct { USINT R:1;   INT A:15; USINT C:1;   INT B:15; };
    struct { USINT r:1; USINT d:2;   SINT p:8; USINT i:7; USINT j:7; USINT k:7; };
  } var_t, *pvar_t;
  #pragma pack(pop)
  
  // Получаем массив сеток по дескриптору  
  TGRID *Grids = (TGRID *)(HGR);
  
  if (IX == 0xFF) { // Направление не задано  - заполнение ячеек узла шаблоном TV
  
    for (short int k=0; k < OFF.B; k++) {
      Grids[PGR].A.table[OFF.A+k] = TV;
    }    
    
  } else {          //  Направление задано =>
    if (IX == 0) {    // Главная ячейка (IX == 0)
      Grids[PGR].A.table[OFF.A] = TV;
      /*
      pvar_t pDest = (var_t *) &Grids[PGR].A.table[OFF.A];
      pvar_t pvar  = (var_t *) &TV;
      if (pvar->r) *pDest = *pvar;
      else {
        // if (pvar->A != -16384) 
          pDest->A = pvar->A;
          
        // if (pvar->B != -16384) 
          pDest->B = pvar->B;
          
        pDest->C = pvar->C;
      }
      */
    } else {          // Смежная ячейка (IX > 0)
    
      // В смежных ячейках могут быть только ссылки или воздух (-1)
      // ASSERT(1,NULL,((pvar_t)&TV)->r,TERROR__E_FAIL, 
        //__STRING_LITERAL(29,"it_var_set: Reference wanted!"));
      
      pvar_t pDest = NULL;
      for (short int k=1; k < OFF.B; k++) {
        pvar_t pvar = (var_t *) &Grids[PGR].A.table[OFF.A+k];
        if ((pDest==NULL && pvar->d==0) || pvar->d == IX) {
          pDest = pvar;
          if (pDest->d == IX) break;
        }
      }
      
      // Ячейка должна найтись!!!
      //ASSERT(1,NULL,pDest!=NULL,TERROR__E_FAIL,
        //_STRING_LITERAL(26, "it_var_set: Cell not found!"));
        
      //if (pDest!=NULL) {
        pDest->tv = TV; 
        pDest->d  = IX;  // Значение IX перезаписывается
      //}
    }
  }
  SET_VAR = PGR;
}}

          
END_FUNCTION

(* Лок->Абс координаты *)
FUNCTION Sh_Loc2Abs : TPoint
  VAR_INPUT
    Sh : TShape;  (* Фигура элемента *)
    X : REAL := 0.0;  (* Точка, координата X (loc) *)
    Y : REAL := 0.0;  (* Точка, координата Y (loc) *)
    Z : REAL := 0.0;  (* Точка, координата Z (loc) *)
  END_VAR
  VAR
    Ax : USINT := 0;  (* Направление оси *)
    A : TPoint := [0.0, 0.0, 0.0];  (* Точка в координатах элемента *)
    B : TPoint := [0.0, 0.0, 0.0];  (* Вспомогательная точка *)
    O : TAxO;  (* Индексы координат x, y, z *)
  END_VAR

            (*Sh := get_sh(PIT);*)
Ax := sh_get_ax(Sh);

A := _point(X,Y,Z); 
if (Ax > 0) then 
  (* Цилиндр -> Декарт *)
  O := AxO(Ax);
  A[O.y] := radi(A[O.y]); (* град -> радианы *)
  B[O.x] := A[O.x]*cos(A[O.y]);
  B[O.y] := A[O.x]*sin(A[O.y]);
  B[O.z] := A[O.z];
else 
  B := A;
end_if;
Sh_Loc2Abs := _point(B[0]+Sh.P0[0],B[1]+Sh.P0[1],B[2]+Sh.P0[2]); 




          
END_FUNCTION

(* Точка по индексам узла *)
FUNCTION Sh_Dot2Point : TPoint
  VAR_INPUT
    Sh : TShape;  (* Фигура элемента *)
    I : INT := 0;  (* Индекс узла решетки I *)
    J : INT := 0;  (* Индекс узла решетки J *)
    K : INT := 0;  (* Индекс узла решетки K *)
    bAbs : BOOL := TRUE;  (* Флаг перевода в абс координаты *)
  END_VAR
  VAR
    Hn : TPoint := [0.0, 0.0, 0.0];  (* Шаг сетки *)
    Ax : USINT := 0;  (* Направление оси *)
    Ang : REAL := 0.0;  (* Угловая координата *)
    Ox : TAxO;  (* Индексы координат x, y, z *)
    P : TPoint := [0.0, 0.0, 0.0];  (* Результат деформации *)
  END_VAR

            Ax := sh_get_ax(Sh);

(* (1) Определение локальной точки X, Y, Z  *)
if (Sh.Kn[0]>1) then Hn[0]:=(Sh.Lx[0]/INT_TO_REAL(Sh.Kn[0]-1)); end_if;
if (Sh.Kn[1]>1) then Hn[1]:=(Sh.Lx[1]/INT_TO_REAL(Sh.Kn[1]-1)); end_if;
if (Sh.Kn[2]>1) then Hn[2]:=(Sh.Lx[2]/INT_TO_REAL(Sh.Kn[2]-1)); end_if;

Sh_Dot2Point := _point( 
  Sh.pL[0] + INT_TO_REAL(I) * Hn[0],
  Sh.pL[1] + INT_TO_REAL(J) * Hn[1],
  Sh.pL[2] + INT_TO_REAL(K) * Hn[2] 
);

(* (2) Коррекция точки при изменении формы  *)
if (Ax<>0) then
  Ox := AxO(Ax, true);
  P := Reform(Sh.wF, Sh_Dot2Point[Ox.y], 
                Sh_Dot2Point[Ox.x], Sh.pL[Ox.x], Sh.Lx[Ox.x]);
  Sh_Dot2Point[Ox.x] := P[0];
end_if;

(* Преобразование локальной точки в абсолют *)
if (bAbs) then
  Sh_Dot2Point := 
    Sh_Loc2Abs(Sh, Sh_Dot2Point[0], Sh_Dot2Point[1], Sh_Dot2Point[2]);
end_if;
          
END_FUNCTION

(* Задание значения типа TVar *)
FUNCTION _ref : TVar
  VAR_INPUT
    PIT : SINT := -1;  (* Позиция элемента ссылки *)
    DOT : TDot;  (* Узел решетки *)
    DIR : USINT := 0;  (* Индекс направления [0,1,2,3] *)
  END_VAR

            {{
  #pragma pack(push, 4)
  union { // 32-бит (4 байта)
    TVAR tv;
    struct {  // Значение (var)
      USINT  R:1;       // Флаг R (для var = 0)
        INT  A:15;      // Значение A (актуальное)
      USINT  C:1;       // Флаг C (1-расчёт готов)
        INT  B:15;      // Значение B (предыдущее)
    };
    struct {  // Ссылка   (ref)
      USINT  r:1;       // Флаг r (для ref = 1)
      USINT  d:2;       // Направление (0,1,2,3)
      USINT  p:8;       // Позиция элемента
      USINT  i:7;       // Индекс сетки по DOT (0..127)
      USINT  j:7;       // Индекс сетки по J (0..127)
      USINT  k:7;       // Индекс сетки по K (0..127)
    };
  } var /*= {0}*/;
  #pragma pack(pop)
  var.r=1;              // Флаг r = 1
  var.d=DIR;            // Индекс направления     (d)
  var.p=PIT;            // Ссылка на элемент      (p)
  var.i=DOT.A.table[0]; // Индексы узла элемента  (i)
  var.j=DOT.A.table[1]; // Индексы узла элемента  (j)
  var.k=DOT.A.table[2]; // Индексы узла элемента  (k)
  _REF=var.tv;
}}

          
END_FUNCTION

(* Линк узла сетки с узлом элем. модели *)
FUNCTION link_var : TDot
  VAR_INPUT
    HGR : THandle := 0;  (* Дескриптор массива сеток *)
    PGR : TPos8 := -1;  (* Позиция сетки *)
    Sh : TShape;  (* Фигура элемента *)
    I : INT := 0;  (* Индекс, координата X (loc, Ax) *)
    J : INT := 0;  (* Индекс, координата Y (loc, Ax) *)
    K : INT := 0;  (* Индекс, координата Z (loc, Ax) *)
    Ix : USINT := 0;  (* Направление оси (0-нет, 1-Ox, 2-Oy, 3-Oz) *)
    ign : TPos8 := -1;  (* Позиция игнорируемого элемента *)
    Dx : REAL := 0.1;  (* Смещение "сверла" за грань *)
    Dyz : REAL := 0.1;  (* Смещение "сверла" внутрь грани *)
  END_VAR
  VAR
    Mx : REAL := 0.0;  (* Множитель смещения по X *)
    My : REAL := 0.0;  (* Множитель смещения по Y *)
    Mz : REAL := 0.0;  (* Множитель смещения по Z *)
    Pt : TPoint := [0.0, 0.0, 0.0];  (* Точка анализа *)
    Dot : TDot;  (* Результат проверки точки *)
  END_VAR

            if (Ix <> 0) then (* при линковке узлов смежных элементов *)

  (* Находим точку в данном узле решётки (лок) *)
  Pt  := Sh_Dot2Point(Sh, I, J, K, false);

  (* "Сверлим стену" *)
  if (I=0) then Mx:=1.0; elsif (I=Sh.Kn[0]-1) then Mx:=-1.0; end_if;
  if (J=0) then My:=1.0; elsif (J=Sh.Kn[1]-1) then My:=-1.0; end_if;
  if (K=0) then Mz:=1.0; elsif (K=Sh.Kn[2]-1) then Mz:=-1.0; end_if;
  
  case Ix of
    1: Pt := _point(Pt[0]-Mx*Dx , Pt[1]+My*Dyz, Pt[2]+Mz*Dyz);
    2: Pt := _point(Pt[0]+Mx*Dyz, Pt[1]-My*Dx , Pt[2]+Mz*Dyz);
    3: Pt := _point(Pt[0]+Mx*Dyz, Pt[1]+My*Dyz, Pt[2]-Mz*Dx );
  end_case;
  
  (* Преобразование локальной точки в абсолют *)
  Pt := Sh_Loc2Abs(Sh, Pt[0], Pt[1], Pt[2]);

else (* при линковке узлов составных элементов и поверхностей *)

  (* Находим точку в данном узле решётки (абс) *)
  Pt := Sh_Dot2Point(Sh, I, J, K);

end_if;

(* Находим элемент, содержащий эту точку *)
Dot := Do_FindDot(Pt[0], Pt[1], Pt[2], ign);

(* Заносим ссылку на найденный элемент в сетку *)
PGR := set_var( HGR, PGR, 
  knoff(Sh.Kn[0], Sh.Kn[1], Sh.Kn[2], I,J,K), 
  _ref(int_to_sint(Dot.v), Dot), 
  Ix 
);

(* Возвращаем позицию сетки, если слинковано, иначе = -1 *)
link_var := (Dot);

          
END_FUNCTION

(* Направление оси симметрии *)
FUNCTION sh_set_ax : TShape
  VAR_INPUT
    SH : TShape;  (* Фигура элемента *)
    Ax : USINT;  (* Направление оси *)
  END_VAR

            Sh.wF := Sh.wF or shl(USINT_TO_WORD(Ax), 12);
sh_set_ax := Sh;
          
END_FUNCTION

(* Состояние элемента (общее) *)
FUNCTION set_cn : TPos8
  VAR_INPUT
    PIT : TPos8 := -1;  (* Позиция элемента *)
    COND : TCond;  (* Состояние элемента *)
  END_VAR

            {{ 
  __GET_GLOBAL_ITS()->CN.table[PIT] = COND;
  return (SET_CN = PIT);
}}

          
END_FUNCTION

(* Сборка состояния узла *)
FUNCTION _cond : TCond
  VAR_INPUT
    ID : UINT := 0;  (* ID элемента *)
    Tmid : INT := -1;  (* Средняя температура *)
    Tmin : TDot;  (* Минимальная температура *)
    Tmax : TDot;  (* Максимальная температура *)
  END_VAR

            _COND.ID   := ID;
_COND.TMID := TMID;
_COND.TMIN := TMIN;
_COND.TMAX := TMAX;

          
END_FUNCTION

(* Состояние элемента (общее) *)
FUNCTION get_cn : TCond
  VAR_INPUT
    PIT : TPos8 := -1;  (* Позиция элемента *)
  END_VAR

            {{ 
  return (GET_CN = 
    (
      (PIT != -1) ? 
      __GET_GLOBAL_ITS()->CN.table[PIT] 
      : _COND(1, NULL, 0, 2000, _DOT(1,NULL,2000,0,0,0), _DOT(1,NULL,2000,0,0,0))
    )
  ); 
}}

          
END_FUNCTION

(* Записывает копию элемента *)
FUNCTION set_it : TPos8
  VAR_INPUT
    PIT : TPos8 := -1;  (* Позиция элемента *)
    ITEM : TItem;  (* Новый элемент *)
  END_VAR

            {{ return (SET_IT = ( __GET_GLOBAL_ITS()->IT.table[PIT] = ITEM, PIT) ); }}

          
END_FUNCTION

(* Выдаёт копию элемента *)
FUNCTION get_it : TItem
  VAR_INPUT
    PIT : TPos8 := -1;  (* Позиция элемента *)
  END_VAR

            {{ return (GET_IT = __GET_GLOBAL_ITS()->IT.table[PIT]); }}

          
END_FUNCTION

(* Возвращает фигуру элемента *)
FUNCTION set_sh : TPos8
  VAR_INPUT
    PSH : TPos8 := -1;  (* Позиция фигуры элемента *)
    Shape : TShape;  (* Фигура элемента *)
  END_VAR

            {{ return (SET_SH = ( __GET_GLOBAL_ITS()->SH.table[PSH] = SHAPE, PSH) ); }}

          
END_FUNCTION

(* Сборка фигуры поверхности *)
FUNCTION _surf : TShape
  VAR_INPUT
    PIT : TPos8 := -1;  (* Позиция элемента *)
    Ax : USINT := 0;  (* Направление перпендикуляра [0..2] *)
    X : REAL := 0.0;  (* Координата X точки привязки *)
    Y : REAL := 0.0;  (* Координата Y точки привязки *)
    Z : REAL := 0.0;  (* Координата Z точки привязки *)
  END_VAR
  VAR
    Pt : TPoint := [0.0, 0.0, 0.0];  (* Точка *)
  END_VAR

            (* Наследуем фигуру элемента модели *)
if (PIT < 0) then PIT := 0; end_if;
_surf := get_sh(PIT);

(* Уточняем размерность сетки [64x64] *)
_surf.wF := 0;
_surf.Kn := _knot(64,64,64);
_surf.Kn[Ax] := 1;

(* Уточняем положение по точке привязки *)
Pt := _point(X,Y,Z);
(*
_surf.pL[0] := _surf.pL[0]+0.1;
_surf.pL[1] := _surf.pL[1]+0.1;
_surf.pL[2] := _surf.pL[2]+0.1;
*)
_surf.pL[Ax] := Pt[Ax]; (* смещение по координате Ax *)
(*
_surf.Lx[0] := _surf.Lx[0]-0.2;
_surf.Lx[1] := _surf.Lx[1]-0.2;
_surf.Lx[2] := _surf.Lx[2]-0.2;
*)
_surf.Lx[Ax] := 0.0;    (* размер плоскости по Ax =0 *)
          
END_FUNCTION

(* Заголовок модели *)
FUNCTION get_h : THead
  VAR_INPUT
    Dummy : DINT := 0;
  END_VAR

            {{ return (GET_H = *__GET_GLOBAL_HDR()); }}
          
END_FUNCTION

(* Профиль величины *)
FUNCTION get_pr : TProf
  VAR_INPUT
    PPR : TPos8 := -1;  (* Позиция профиля *)
  END_VAR

            {{ return (GET_PR = __GET_GLOBAL_STS()->PR.table[PPR]); }}

          
END_FUNCTION

(* Буферная величина *)
FUNCTION get_bf : REAL
  VAR_INPUT
    PBF : TPos16 := -1;  (* Позиция в буфере *)
  END_VAR

            {{ return (GET_BF = __GET_GLOBAL_STS()->BF.table[PBF]); }}

          
END_FUNCTION

(* Связанная величина *)
FUNCTION get_vl : TVal
  VAR_INPUT
    PVL : TPos8 := -1;  (* Позиция величины *)
  END_VAR

            {{ return (GET_VL = __GET_GLOBAL_STS()->VL.table[PVL]); }}

          
END_FUNCTION

(* Материал элемента *)
FUNCTION get_mt : TMat
  VAR_INPUT
    PMT : TPos8 := -1;  (* Позиция материала *)
  END_VAR

            {{ return (GET_MT = __GET_GLOBAL_STS()->MT.table[PMT]); }}

          
END_FUNCTION

(* Время расчёта по направлению Ix *)
FUNCTION get_pdt : DT
  VAR_INPUT
    PIT : TPos8 := -1;  (* Позиция элемента *)
    Ix : USINT := 0;  (* Направление расчёта *)
  END_VAR

            {{ return (GET_PDT = __GET_GLOBAL_ITS()->IT.table[PIT].PDT.table[IX]); }}

          
END_FUNCTION

(* Задать время расчёта *)
FUNCTION set_pdt : TPos8
  VAR_INPUT
    PIT : TPos8 := -1;  (* Позиция элемента *)
    Ix : USINT := 0;  (* Направление расчёта *)
    CDT : DT := DT#2000-01-01-00:00:00;  (* Текущее время *)
  END_VAR

            {{ return (SET_PDT = (__GET_GLOBAL_ITS()->IT.table[PIT].PDT.table[IX] = CDT, PIT)); }}

          
END_FUNCTION

(* Индекс материала *)
FUNCTION it_im : TPos8
  VAR_INPUT
    PIT : TPos8 := -1;  (* Позиция элемента *)
  END_VAR

            {{ return (IT_IM = __GET_GLOBAL_ITS()->IT.table[PIT].IM); }}

          
END_FUNCTION

(* Индекс величины *)
FUNCTION it_iv : TPos8
  VAR_INPUT
    PIT : TPos8 := -1;  (* Позиция элемента *)
  END_VAR

            {{ return (IT_IV = __GET_GLOBAL_ITS()->IT.table[PIT].IV); }}

          
END_FUNCTION

(* Задание значения типа TVar *)
FUNCTION get_var : TVar
  VAR_INPUT
    HGR : THandle := 0;  (* Дескриптор массива сеток *)
    PGR : TPos8 := -1;  (* Позиция сетки в массиве *)
    OFF : P_INT;  (* Смещение узла в сетке *)
    IX : USINT := 0;  (* Ключ направления (0xff-неопределён) *)
  END_VAR

            {{
  #pragma pack(push, 4)
  typedef union {
    TVAR tv;
    struct { USINT R:1;   INT A:15; USINT C:1;   INT B:15; };
    struct { USINT r:1; USINT d:2;   SINT p:8; USINT i:7; USINT j:7; USINT k:7; };
  } var_t, *pvar_t;
  #pragma pack(pop)

  // Получаем массив сеток по дескриптору  
  TGRID *Grids = (TGRID *)(HGR);
  
  if (IX == 0) {        // Главная ячейка узла
  
    GET_VAR = Grids[PGR].A.table[OFF.A];
    
  } else if (IX < 4) {  // Смежная ячейка узла
  
    for (int k=(GET_VAR=(TVAR)0, 1); k < OFF.B; k++) {
      GET_VAR = Grids[PGR].A.table[OFF.A+k];
      if (((pvar_t)&GET_VAR)->d == IX) break;
    }
    
    // Значение смежных ячеек может быть только ссылочным (!)
    // ASSERT(1, NULL, ((pvar_t)&GET_VAR)->r, TERROR__E_FAIL, 
      //__STRING_LITERAL(29,"GET_VAR: Reference wanted!"));
      
  } else {

    // Неверное значение IX
    // ASSERT(1, NULL, FALSE, TERROR__E_FAIL, 
      //__STRING_LITERAL(29,"GET_VAR: Invalid IX!"));
  
  }
}}

          
END_FUNCTION

(* Значение поля 'p' структуры var *)
FUNCTION var_up : TVar
  VAR_INPUT
    TV : TVar := 0;  (* Структура типа TVar *)
  END_VAR

            {{
  #pragma pack(push, 4)
  typedef union {
    TVAR tv;
    struct { USINT R:1;   INT A:15; USINT C:1;   INT B:15; };
    struct { USINT r:1; USINT d:2;   SINT p:8; USINT i:7; USINT j:7; USINT k:7; };
  } var_t, *pvar_t;
  #pragma pack(pop)
  pvar_t pvar = (pvar_t)&TV;
  // Если значение не ссылка - "поднимаем" значение A->B!
  if (!pvar->r) {
    //if (pvar->C) 
      pvar->B = (pvar->C=0, pvar->A);
  }
  VAR_UP = TV;
}}

          
END_FUNCTION

(* Средняя температура элемента *)
FUNCTION cn_mid : INT
  VAR_INPUT
    Cond : TCond;  (* Состояние элемента *)
  END_VAR

            CN_MID := COND.TMID;

          
END_FUNCTION

(* TRUE, если элемент - родитель *)
FUNCTION is_parent : BOOL
  VAR_INPUT
    PIT : TPos8 := -1;  (* Позиция элемента *)
  END_VAR

            {{ return (IS_PARENT = (__GET_GLOBAL_ITS()->IT.table[PIT].NUM > 0)); }}

          
END_FUNCTION

(* TRUE, если СК - цилиндрическая *)
FUNCTION is_cyl : BOOL
  VAR_INPUT
    PIT : TPos8 := -1;  (* Позиция элемента *)
  END_VAR

            IS_CYL := (sh_get_ax(get_sh(PIT)) <> 0);

          
END_FUNCTION

(* Идентификатор элемента *)
FUNCTION it_id : UINT
  VAR_INPUT
    PIT : TPos8 := -1;  (* Позиция элемента *)
  END_VAR

            {{ return (IT_ID = __GET_GLOBAL_ITS()->IT.table[PIT].ID); }}

          
END_FUNCTION

(* Валидация позиции элемента *)
FUNCTION it_pos : TPos8
  VAR_INPUT
    PIT : TPos8 := -1;  (* Позиция элемента *)
    bForce : BOOL := false;  (* Усиленная проверка *)
  END_VAR

            {{ 
  if (BFORCE) {
    ASSERT(1, NULL, 
     (PIT >= 0) && (PIT < __GET_GLOBAL_HDR()->NI), TERROR__E_ITEMPOS, __INIT_STRING);
  }
  return (IT_POS = ( (PIT < 0) || (PIT >= __GET_GLOBAL_HDR()->NI) ? (0) : PIT ));
}}

          
END_FUNCTION

(* Установка статуса *)
FUNCTION st_set_stat : BOOL
  VAR_INPUT
    err : TError := E_SUCCESS;  (* Код ошибки *)
    par : UINT := 0;  (* Параметр состояния *)
    str : STRING := '';  (* Строка состояния *)
  END_VAR

            {{ 
  __GET_GLOBAL_STAT()->ERR=ERR; 
  __GET_GLOBAL_STAT()->PAR=PAR; 
  __GET_GLOBAL_STAT()->STR=STR;
  LOGMSG(1,NULL,STR,LOGLEVEL__DEBUG,ERR);
  return (ST_SET_STAT=ST_CHECK(1,NULL,FALSE));
}}

          
END_FUNCTION

(* Процессор перед расчётом модели *)
FUNCTION Do_PreProc : BOOL
  VAR_INPUT
    PIT : TPos8 := -1;  (* Начальная позиция *)
  END_VAR
  VAR
    It : TIter;  (* Итератор *)
  END_VAR

            Do_PreProc := st_check(false);
if (not Do_PreProc) then return; end_if;

(* Обход дерева элементов *)
Do_PreProc := true;
it := it_begin(it_pos(PIT));
while (it.item <>-1) do
  case (it.dir) of
  DIR_UP:
    { }
  end_case;
  it := it_next(it);
end_while;

{ __exit: }
return;

{ __error: } 
Do_PreProc := st_set_stat(E_PREPROC, it_id(it.item));

          
END_FUNCTION

(* Температура -> Код *)
FUNCTION T2C : INT
  VAR_INPUT
    Temp : REAL := 0.0;  (* Температура *)
  END_VAR

            T2C := real_to_int(Temp*100.0);
          
END_FUNCTION

(* Значение поля 'v' структуры var *)
FUNCTION var_v : INT
  VAR_INPUT
    TV : TVar := -1;  (* Структура типа TVar *)
    GET_A : BOOL := true;  (* Возвратить значение "A" *)
  END_VAR
  VAR
    Sh : TShape;  (* Фигура *)
  END_VAR

            {{
  #pragma pack(push, 4)
  typedef union {
    TVAR tv;
    struct { USINT R:1;   INT A:15; USINT C:1;   INT B:15; };
    struct { USINT r:1; USINT d:2;   SINT p:8; USINT i:7; USINT j:7; USINT k:7; };
  } var_t, *pvar_t;
  #pragma pack(pop)
  pvar_t pvar = (pvar_t)&TV;
  
  // Решаем ссылку (если нужно)
  while (pvar->r) {
    if (pvar->p >= 0) {
      // ссылка должна быть реальной (!)
      //ASSERT(1, NULL, (pvar->p < __GET_GLOBAL_HDR()->NI), 
      //  TERROR__E_FAIL, __STRING_LITERAL(22,"var_v: Reference fail!") );
      
      // Переход к элементу по ссылке:
      SH = GET_SH(1, NULL, pvar->p);
      P_INT Off = KNOFF(1, NULL, 
          SH.KN.table[0], SH.KN.table[1], SH.KN.table[2], 
          pvar->i, pvar->j, pvar->k
      );
      pvar = (pvar_t) &__GET_GLOBAL_ITS()->GR.table[pvar->p].A.table[Off.A];
    } else {  
      // элемент не существует -> воздух
      return (VAR_V = 2000); // 20.00 градусов Цельсия
    }
  }
  
  VAR_V = (GET_A) ? pvar->A : pvar->B;
}}

          
END_FUNCTION

(* Обновление значений в узлах сетки *)
FUNCTION it_update : TPos8
  VAR_INPUT
    PIT : TPos8 := -1;  (* Позиция элемента *)
  END_VAR
  VAR
    Pt : TPoint;  (* Точка *)
    Kn : TKnot;  (* Размерность сетки *)
    Sh : TShape;  (* Фигура элемента *)
    Off : P_INT;  (* Смещение узла сетки *)
    iVar : INT := 0;  (* Температура узла сетки *)
    TV : TVar := -1;  (* Значение узла сетки *)
    Tmid : REAL := 0.0;  (* Средняя температура *)
    count : INT := 0;  (* Счётчик узлов при подсчёте *)
    i : INT := 0;  (* Счётчик цикла по координате *)
    j : INT := 0;  (* Счётчик цикла по координате *)
    k : INT := 0;  (* Счётчик цикла по координате *)
    Cond : TCond;  (* Состояние элемента *)
  END_VAR

            Sh := get_sh(it_pos(PIT));
Kn := Sh.Kn;
Cond.Tmin.V := 16383;   (* max_int7 *)
Cond.Tmax.V := -16384;  (* min_int7 *)

(* Вычисление средней, минимальной и максимальной температур *)
for i:=0 to Kn[0]-1 do
  for J:=0 to Kn[1]-1 do
    for K:=0 to Kn[2]-1 do
      Off   := knoff(Kn[0], Kn[1], Kn[2], i,J,K);
      TV    := get_var(its_gr(0), PIT, Off);
      iVar  := var_v(TV);
      
      Tmid  := ( Tmid*int_to_real(count) + (int_to_real(iVar)/100.0) ) / 
                    int_to_real(count+1);
      if (iVar < Cond.Tmin.V) then Cond.Tmin := _dot(iVar, i,j,k); end_if;
      if (iVar > Cond.Tmax.V) then Cond.Tmax := _dot(iVar, i,j,k); end_if;
      
      TV    := var_up(TV);
      PIT   := set_var(its_gr(0), PIT, Off, (TV));
      count := count+1;
    end_for;
  end_for;
end_for;

(* Средняя температура элемента *)
(* Cond.Tmid := T2C(Tmid); *)
{{ COND.TMID = (INT)(TMID * 100.0); }}

(* Минимальная температура элемента *)
Pt := Sh_Dot2Point(Sh, Cond.Tmin.A[0], Cond.Tmin.A[1], Cond.Tmin.A[2]);
Cond.Tmin.A[0] := real_to_int(Pt[0]);
Cond.Tmin.A[1] := real_to_int(Pt[1]);
Cond.Tmin.A[2] := real_to_int(Pt[2]);

(* Максимальная температура элемента *)         
Pt := Sh_Dot2Point(Sh, Cond.Tmax.A[0], Cond.Tmax.A[1], Cond.Tmax.A[2]);
Cond.Tmax.A[0] := real_to_int(Pt[0]);
Cond.Tmax.A[1] := real_to_int(Pt[1]);
Cond.Tmax.A[2] := real_to_int(Pt[2]);

(* Сохраняем состояние элемента *)
PIT := set_cn(PIT, Cond);

{{ // TEST
  if (PIT==53) *__GET_GLOBAL_RTEST() = TMID;
}}

IT_Update := PIT;


          
END_FUNCTION

(* Процессор после расчёта модели *)
FUNCTION Do_PostProc : BOOL
  VAR_INPUT
    PIT : TPos8 := -1;  (* Начальная позиция *)
  END_VAR
  VAR
    It : TIter;  (* Итератор *)
  END_VAR

            (* Проверка статуса программы *)
Do_PostProc := st_check(false);
if (not Do_PostProc) then return; end_if;

(* Обход дерева элементов *)
Do_PostProc := true;
it := it_begin(it_pos(PIT));
while (it.item <>-1) do
  case (it.dir) of
  DIR_UP:
    (* Обновление состояния сетки элемента *)
    it.item := it_update(it.item);
  end_case;
  it := it_next(it);
end_while;

{ __exit: }
return;

{ __error: }
Do_PostProc := st_set_stat(E_POSTPROC, it_id(it.item));


          
END_FUNCTION

(* Код -> Температура *)
FUNCTION C2T : REAL
  VAR_INPUT
    Code : INT := 0;  (* Код температуры *)
  END_VAR

            C2T := int_to_real(Code)/100.0;
          
END_FUNCTION

(* Строка ID в 16# представлении *)
FUNCTION ID2Str : STRING
  VAR_INPUT
    IID : UINT;  (* Идентификатор *)
  END_VAR
  VAR
    i : USINT;  (* Индекс *)
    IDs : ARRAY[0..3] OF USINT;  (* Знаки идентификатора *)
    ch : ARRAY[0..3] OF STRING;  (* Знаки идентификатора *)
  END_VAR

            (* Распаковка идентификатора элемента на отдельные байты *)
IDs[0]  := WORD_TO_USINT(SHR((UINT_TO_WORD(IID) and 16#F000),12));
IDs[1]  := WORD_TO_USINT(SHR((UINT_TO_WORD(IID) and 16#0F00), 8));
IDs[2]  := WORD_TO_USINT(SHR((UINT_TO_WORD(IID) and 16#00F0), 4));
IDs[3]  := WORD_TO_USINT(SHR((UINT_TO_WORD(IID) and 16#000F), 0));
(* Замена цифр на символы *)
for i:=0 to 3 do
  case (IDs[i]-10) of
  0: ch[i]:='A';
  1: ch[i]:='B';
  2: ch[i]:='C';
  3: ch[i]:='D';
  4: ch[i]:='E';
  5: ch[i]:='F';
  else ch[i]:=USINT_TO_STRING(IDs[i]);
  end_case;
end_for;
(* Сборка идентификатора *)
ID2Str := MakeMsg(ch[0], ch[1], ch[2], ch[3]);

          
END_FUNCTION

(* Строка состояния элемента *)
FUNCTION IT_CondStr : STRING
  VAR_INPUT
    PIT : TPos8 := -1;  (* Позиция элемента *)
  END_VAR
  VAR
    Cond : TCond;  (* Состояние элемента *)
    bP : BOOL := FALSE;  (* Флаг 'элемент-родитель' *)
    msg : STRING := '';  (* Строка состояния *)
  END_VAR

            Cond := get_cn(it_pos(PIT));
if (is_poly(PIT)) then
  msg := MakeMsg(msg, ' [', ID2Str(IT_ID(PIT)), ',');
  msg := MakeMsg(msg,       SINT_TO_STRING(PIT), ',');
  msg := MakeMsg(msg, INT_TO_STRING( REAL_TO_INT(C2T(Cond.Tmid)) ), ',');
  (* msg := MakeMsg(msg, INT_TO_STRING( REAL_TO_INT(C2T(Cond.Tmin.V)) ), ']'); *)
  msg := MakeMsg(msg, INT_TO_STRING( REAL_TO_INT(C2T(Cond.Tmax.V)) ), ']');
else 
  msg := MakeMsg(msg, ' (', ID2Str(IT_ID(PIT)), ',');
  msg := MakeMsg(msg,       SINT_TO_STRING(PIT), ',');
  msg := MakeMsg(msg, INT_TO_STRING( REAL_TO_INT(C2T(Cond.Tmid)) ), ',');
  (* msg := MakeMsg(msg, INT_TO_STRING( REAL_TO_INT(C2T(Cond.Tmin.V)) ), ']'); *)
  msg := MakeMsg(msg, INT_TO_STRING( REAL_TO_INT(C2T(Cond.Tmax.V)) ), ')');
end_if;
IT_CondStr:=msg;
          
END_FUNCTION

(* Протокол состояния модели *)
FUNCTION Do_LogCond : BOOL
  VAR_INPUT
    PIT : TPos8 := -1;  (* Начальная позиция *)
  END_VAR
  VAR
    It : TIter;  (* Итератор *)
    msg : STRING := '';  (* Сообщение в протокол *)
    i : SINT := 0;  (* Индекс *)
  END_VAR

            Do_LogCond := st_check(false);
if (not Do_LogCond) then return; end_if;
(* Обход дерева элементов *)
i:=0;
it := it_begin(it_pos(PIT));
while (it.item <>-1) do
  if (len(msg)=0) then msg := MakeMsg(' -> '); end_if;
  case (it.dir) of
  DIR_UP:
    (*if (not it_parent(it.item)) then*) (* состояние терминального элемента *)
      msg := MakeMsg(msg, IT_CondStr(it.item));
      if (mod((i+1),5)=0) then msg:=LogMsg(MakeMsg(msg, ';')); end_if;
      i := i+1;
    (*end_if;*)
  end_case;
  it := it_next(it);
end_while;
if (len(msg)>0) then msg:=LogMsg(MakeMsg(msg, ';')); end_if;
msg:=LogMsg(' --- ');
(*Do_LogCond := true;*)
          
END_FUNCTION

(* "Связывание" элементов на гранях *)
FUNCTION Do_LinkItems : INT
  VAR_INPUT
    PIT : TPos8 := -1;  (* Первичный узел обхода *)
  END_VAR
  VAR
    It : TIter;  (* Итератор *)
    B : BYTE := 0;  (* Флаги граней, контактирующих с воздухом *)
    I : INT := 0;  (* Индекс сетки X *)
    J : INT := 0;  (* Индекс сетки Y *)
    K : INT := 0;  (* Индекс сетки Z *)
    nPos : SINT := 0;  (* Найденный узел *)
    nAir : INT := 0;  (* Количество граней, выходящих на "воздух" *)
    nItems : INT := 0;  (* Количество элементов с контактом с "воздухом" *)
    Sh : TShape;  (* Фигура элемента *)
    Dot : TDot;  (* Результат проверки точки *)
    Pt : TPoint;  (* Точка узла *)
  END_VAR

            Do_LinkItems := (-1);
if (not st_check(false)) then return; end_if;

(* Обход дерева элементов *)
it := it_begin(it_pos(PIT));
while (it.item <> -1) do
  case (it.dir) of
  DIR_UP:
    B     := 0; 
    nAir  := 0;
    Sh := get_sh(it.item);
    
    (* Рассчитываем точки по граням X=(Х0,Kn[0]-1) *)
    for I:=0 to Sh.Kn[0]-1 do
      for J:=0 to Sh.Kn[1]-1 do
        for K:=0 to Sh.Kn[2]-1 do

          if (not is_poly(it.item)) then  
            (* линкуем узлы конечных элементов *)
          
            if (I=0 or I=Sh.Kn[0]-1) then  (* по координате X (Ix=1) *)
              Dot := link_var(its_gr(0), it.item, Sh, I, J, K, 1, it.item);
              if (Dot.v = -1) then   (* Воздух *)
                if (I=0) then B:=(B or shl(16#01, 1)); else B:=(B or shl(16#01, 2)); end_if;
              end_if;
            end_if;
            
            if (J=0 or J=Sh.Kn[1]-1) then  (* по координате Y  (Ix=2) *)
              Dot := link_var(its_gr(0), it.item, Sh, I, J, K, 2, it.item);
              if (Dot.v = -1) then  (* Воздух *)
                if (J=0) then B:=(B or shl(16#01, 3)); else B:=(B or shl(16#01, 4)); end_if;
              end_if;
            end_if;
            
            if (K=0 or K=Sh.Kn[2]-1) then  (* по координате Z  (Ix=3) *)
              Dot := link_var(its_gr(0), it.item, Sh, I, J, K, 3, it.item);
              if (Dot.v = -1) then  (* Воздух *)
                if (K=0) then B:=(B or shl(16#01, 5)); else B:=(B or shl(16#01, 6)); end_if;
              end_if;
            end_if;
            
          else    (* линкуем сетку составного элемента (Ix=0, default) *)
          
            Dot := link_var(its_gr(0), it.item, Sh, I, J, K);
            
          end_if;
          
        end_for;
      end_for;
    end_for;
    
    (* Суммируем количество граней, контактирующих с воздухом *)
    for i:=1 to 6 do
      if ((B and shl(16#01, i)) <> 0) then nAir:=nAir+1; end_if;
    end_for;
      
    (* Подсчёт элеметов, контактирующих с "воздухом" *)
    if (nAir > 0) then nItems := nItems+1; end_if;
    
  end_case;
  it := it_next(it);
end_while;

Do_LinkItems := (nItems);

          
END_FUNCTION

(* Задание значения типа TVar *)
FUNCTION _var : TVar
  VAR_INPUT
    A : INT := -16384;  (* Значение V1 (текущее значение) *)
    B : INT := -16384;  (* Значение V2 (предыдущее значение) *)
    C : BOOL := false;  (* Флаг "расчёт выполнен" *)
  END_VAR

            {{
  #pragma pack(push, 4)
  union { // 32-бит (4 байта)
    TVAR tv;
    struct {  // Значение (var)
      USINT  R:1;     // Флаг R (для var = 0)
        INT  A:15;    // Значение A (актуальное)
      USINT  C:1;     // Флаг C (1-расчёт готов)
        INT  B:15;    // Значение B (предыдущее)
    };
    struct {  // Ссылка   (ref)
      USINT  r:1;     // Флаг r (для ref = 1)
      USINT  d:2;     // Направление (0,1,2,3)
      USINT  p:8;     // Позиция элемента
      USINT  i:7;     // Индекс сетки по I (0..127)
      USINT  j:7;     // Индекс сетки по J (0..127)
      USINT  k:7;     // Индекс сетки по K (0..127)
    };
  } var = {0};
  #pragma pack(pop)
  
  var.A = A;  // Значение A (текущее)
  var.B = B;  // Значение B (предыдущее)
  var.C = C;  // Флаг "расчёт выполнен" (A!=B)
  
  _VAR = var.tv;
}}

          
END_FUNCTION

(* Установка Temp во всех узлах *)
FUNCTION IT_InitTemp : TPos8
  VAR_INPUT
    PIT : TPos8 := 0;  (* Позиция элемента *)
    Temp : REAL := 0.0;  (* Температура элемента *)
    CLR : BOOL := false;  (* Флаг очистки связей *)
  END_VAR
  VAR
    Sh : TShape;  (* Фигура элемента *)
    I : INT := 0;  (* Счётчик Ix *)
    J : INT := 0;  (* Счётчик Iy *)
    K : INT := 0;  (* Счётчик Iz *)
    M : INT := 0;  (* Счётчик узла *)
    Off : P_INT;  (* Сдвиг узла в массиве *)
  END_VAR

            Sh := get_sh(it_pos(PIT));
for I:=0 to Sh.Kn[0]-1 do
  for J:=0 to Sh.Kn[1]-1 do
    for K:=0 to Sh.Kn[2]-1 do
      Off := knoff(Sh.Kn[0], Sh.Kn[1], Sh.Kn[2], I,J,K);
      if (CLR) then PIT := set_var(its_gr(0), PIT, Off, 0, 16#ff); end_if;
      PIT := set_var(its_gr(0), PIT, Off, _var(T2C(Temp), T2C(Temp)));
    end_for;
  end_for;
end_for;
IT_InitTemp := PIT;

          
END_FUNCTION

(* Индекс (позиция) родителя *)
FUNCTION it_ip : TPos8
  VAR_INPUT
    PIT : TPos8 := -1;  (* Позиция элемента *)
  END_VAR

            {{ return (IT_IP = __GET_GLOBAL_ITS()->IT.table[PIT].PAR); }}

          
END_FUNCTION

(* Компоновка определения элемента *)
FUNCTION m_def : TDef
  VAR_INPUT
    MW0 : UINT;
    MW1 : UINT;
    MW2 : UINT;
    MW3 : UINT;
    MW4 : UINT;
    MW5 : UINT;
    MW6 : UINT;
    MW7 : UINT;
    MW8 : UINT;
    MW9 : UINT;
  END_VAR

            (* Идентификатор, флаги и радиус *)
m_def.ID    := MW0;
m_def.CF    := UINT_TO_WORD(MW1);
m_def.R0    := UINT_TO_INT (MW2);

(* Определение точки начала отсчёта *)
m_def.XYZ[0]:= UINT_TO_INT (MW3);
m_def.XYZ[1]:= UINT_TO_INT (MW4);
m_def.XYZ[2]:= UINT_TO_INT (MW5);

(* Определение габаритов элемента   *)
m_def.LWH[0]:= UINT_TO_INT (MW6);
m_def.LWH[1]:= UINT_TO_INT (MW7);
m_def.LWH[2]:= UINT_TO_INT (MW8);

(* Определение индексов элемента   *)
m_def.Ig    := UINT_TO_SINT((MW9/256)/16);
m_def.Im    := UINT_TO_SINT(mod((MW9/256),16));
m_def.Iv    := UINT_TO_SINT(mod(MW9, 256));

          
END_FUNCTION

(* Чтение определения из регистров *)
FUNCTION_BLOCK GetDef
  VAR_EXTERNAL
    MW0 : UINT;
    MW1 : UINT;
    MW2 : UINT;
    MW3 : UINT;
    MW4 : UINT;
    MW5 : UINT;
    MW6 : UINT;
    MW7 : UINT;
    MW8 : UINT;
    MW9 : UINT;
    MW10 : UINT;
    MW11 : UINT;
    MW12 : UINT;
    MW13 : UINT;
    MW14 : UINT;
    MW15 : UINT;
    MW16 : UINT;
    MW17 : UINT;
    MW18 : UINT;
    MW19 : UINT;
    MW20 : UINT;
    MW21 : UINT;
    MW22 : UINT;
    MW23 : UINT;
    MW24 : UINT;
    MW25 : UINT;
    MW26 : UINT;
    MW27 : UINT;
    MW28 : UINT;
    MW29 : UINT;
    MW30 : UINT;
    MW31 : UINT;
    MW32 : UINT;
    MW33 : UINT;
    MW34 : UINT;
    MW35 : UINT;
    MW36 : UINT;
    MW37 : UINT;
    MW38 : UINT;
    MW39 : UINT;
    MW40 : UINT;
    MW41 : UINT;
    MW42 : UINT;
    MW43 : UINT;
    MW44 : UINT;
    MW45 : UINT;
    MW46 : UINT;
    MW47 : UINT;
    MW48 : UINT;
    MW49 : UINT;
    MW50 : UINT;
    MW51 : UINT;
    MW52 : UINT;
    MW53 : UINT;
    MW54 : UINT;
    MW55 : UINT;
    MW56 : UINT;
    MW57 : UINT;
    MW58 : UINT;
    MW59 : UINT;
    MW60 : UINT;
    MW61 : UINT;
    MW62 : UINT;
    MW63 : UINT;
    MW64 : UINT;
    MW65 : UINT;
    MW66 : UINT;
    MW67 : UINT;
    MW68 : UINT;
    MW69 : UINT;
    MW70 : UINT;
    MW71 : UINT;
    MW72 : UINT;
    MW73 : UINT;
    MW74 : UINT;
    MW75 : UINT;
    MW76 : UINT;
    MW77 : UINT;
    MW78 : UINT;
    MW79 : UINT;
    MW80 : UINT;
    MW81 : UINT;
    MW82 : UINT;
    MW83 : UINT;
    MW84 : UINT;
    MW85 : UINT;
    MW86 : UINT;
    MW87 : UINT;
    MW88 : UINT;
    MW89 : UINT;
    MW90 : UINT;
    MW91 : UINT;
    MW92 : UINT;
    MW93 : UINT;
    MW94 : UINT;
    MW95 : UINT;
    MW96 : UINT;
    MW97 : UINT;
    MW98 : UINT;
    MW99 : UINT;
    MW100 : UINT;
    MW101 : UINT;
    MW102 : UINT;
    MW103 : UINT;
    MW104 : UINT;
    MW105 : UINT;
    MW106 : UINT;
    MW107 : UINT;
    MW108 : UINT;
    MW109 : UINT;
    MW110 : UINT;
    MW111 : UINT;
    MW112 : UINT;
    MW113 : UINT;
    MW114 : UINT;
    MW115 : UINT;
    MW116 : UINT;
    MW117 : UINT;
    MW118 : UINT;
    MW119 : UINT;
    MW120 : UINT;
    MW121 : UINT;
    MW122 : UINT;
    MW123 : UINT;
    MW124 : UINT;
    MW125 : UINT;
    MW126 : UINT;
    MW127 : UINT;
    MW128 : UINT;
    MW129 : UINT;
    MW130 : UINT;
    MW131 : UINT;
    MW132 : UINT;
    MW133 : UINT;
    MW134 : UINT;
    MW135 : UINT;
    MW136 : UINT;
    MW137 : UINT;
    MW138 : UINT;
    MW139 : UINT;
    MW140 : UINT;
    MW141 : UINT;
    MW142 : UINT;
    MW143 : UINT;
    MW144 : UINT;
    MW145 : UINT;
    MW146 : UINT;
    MW147 : UINT;
    MW148 : UINT;
    MW149 : UINT;
    MW150 : UINT;
    MW151 : UINT;
    MW152 : UINT;
    MW153 : UINT;
    MW154 : UINT;
    MW155 : UINT;
    MW156 : UINT;
    MW157 : UINT;
    MW158 : UINT;
    MW159 : UINT;
    MW160 : UINT;
    MW161 : UINT;
    MW162 : UINT;
    MW163 : UINT;
    MW164 : UINT;
    MW165 : UINT;
    MW166 : UINT;
    MW167 : UINT;
    MW168 : UINT;
    MW169 : UINT;
    MW170 : UINT;
    MW171 : UINT;
    MW172 : UINT;
    MW173 : UINT;
    MW174 : UINT;
    MW175 : UINT;
    MW176 : UINT;
    MW177 : UINT;
    MW178 : UINT;
    MW179 : UINT;
    MW180 : UINT;
    MW181 : UINT;
    MW182 : UINT;
    MW183 : UINT;
    MW184 : UINT;
    MW185 : UINT;
    MW186 : UINT;
    MW187 : UINT;
    MW188 : UINT;
    MW189 : UINT;
    MW190 : UINT;
    MW191 : UINT;
    MW192 : UINT;
    MW193 : UINT;
    MW194 : UINT;
    MW195 : UINT;
    MW196 : UINT;
    MW197 : UINT;
    MW198 : UINT;
    MW199 : UINT;
    MW200 : UINT;
    MW201 : UINT;
    MW202 : UINT;
    MW203 : UINT;
    MW204 : UINT;
    MW205 : UINT;
    MW206 : UINT;
    MW207 : UINT;
    MW208 : UINT;
    MW209 : UINT;
    MW210 : UINT;
    MW211 : UINT;
    MW212 : UINT;
    MW213 : UINT;
    MW214 : UINT;
    MW215 : UINT;
    MW216 : UINT;
    MW217 : UINT;
    MW218 : UINT;
    MW219 : UINT;
    MW220 : UINT;
    MW221 : UINT;
    MW222 : UINT;
    MW223 : UINT;
    MW224 : UINT;
    MW225 : UINT;
    MW226 : UINT;
    MW227 : UINT;
    MW228 : UINT;
    MW229 : UINT;
    MW230 : UINT;
    MW231 : UINT;
    MW232 : UINT;
    MW233 : UINT;
    MW234 : UINT;
    MW235 : UINT;
    MW236 : UINT;
    MW237 : UINT;
    MW238 : UINT;
    MW239 : UINT;
    MW240 : UINT;
    MW241 : UINT;
    MW242 : UINT;
    MW243 : UINT;
    MW244 : UINT;
    MW245 : UINT;
    MW246 : UINT;
    MW247 : UINT;
    MW248 : UINT;
    MW249 : UINT;
    MW250 : UINT;
    MW251 : UINT;
    MW252 : UINT;
    MW253 : UINT;
    MW254 : UINT;
    MW255 : UINT;
    MW256 : UINT;
    MW257 : UINT;
    MW258 : UINT;
    MW259 : UINT;
    MW260 : UINT;
    MW261 : UINT;
    MW262 : UINT;
    MW263 : UINT;
    MW264 : UINT;
    MW265 : UINT;
    MW266 : UINT;
    MW267 : UINT;
    MW268 : UINT;
    MW269 : UINT;
    MW270 : UINT;
    MW271 : UINT;
    MW272 : UINT;
    MW273 : UINT;
    MW274 : UINT;
    MW275 : UINT;
    MW276 : UINT;
    MW277 : UINT;
    MW278 : UINT;
    MW279 : UINT;
    MW280 : UINT;
    MW281 : UINT;
    MW282 : UINT;
    MW283 : UINT;
    MW284 : UINT;
    MW285 : UINT;
    MW286 : UINT;
    MW287 : UINT;
    MW288 : UINT;
    MW289 : UINT;
    MW290 : UINT;
    MW291 : UINT;
    MW292 : UINT;
    MW293 : UINT;
    MW294 : UINT;
    MW295 : UINT;
    MW296 : UINT;
    MW297 : UINT;
    MW298 : UINT;
    MW299 : UINT;
    MW300 : UINT;
    MW301 : UINT;
    MW302 : UINT;
    MW303 : UINT;
    MW304 : UINT;
    MW305 : UINT;
    MW306 : UINT;
    MW307 : UINT;
    MW308 : UINT;
    MW309 : UINT;
    MW310 : UINT;
    MW311 : UINT;
    MW312 : UINT;
    MW313 : UINT;
    MW314 : UINT;
    MW315 : UINT;
    MW316 : UINT;
    MW317 : UINT;
    MW318 : UINT;
    MW319 : UINT;
    MW320 : UINT;
    MW321 : UINT;
    MW322 : UINT;
    MW323 : UINT;
    MW324 : UINT;
    MW325 : UINT;
    MW326 : UINT;
    MW327 : UINT;
    MW328 : UINT;
    MW329 : UINT;
    MW330 : UINT;
    MW331 : UINT;
    MW332 : UINT;
    MW333 : UINT;
    MW334 : UINT;
    MW335 : UINT;
    MW336 : UINT;
    MW337 : UINT;
    MW338 : UINT;
    MW339 : UINT;
    MW340 : UINT;
    MW341 : UINT;
    MW342 : UINT;
    MW343 : UINT;
    MW344 : UINT;
    MW345 : UINT;
    MW346 : UINT;
    MW347 : UINT;
    MW348 : UINT;
    MW349 : UINT;
    MW350 : UINT;
    MW351 : UINT;
    MW352 : UINT;
    MW353 : UINT;
    MW354 : UINT;
    MW355 : UINT;
    MW356 : UINT;
    MW357 : UINT;
    MW358 : UINT;
    MW359 : UINT;
    MW360 : UINT;
    MW361 : UINT;
    MW362 : UINT;
    MW363 : UINT;
    MW364 : UINT;
    MW365 : UINT;
    MW366 : UINT;
    MW367 : UINT;
    MW368 : UINT;
    MW369 : UINT;
    MW370 : UINT;
    MW371 : UINT;
    MW372 : UINT;
    MW373 : UINT;
    MW374 : UINT;
    MW375 : UINT;
    MW376 : UINT;
    MW377 : UINT;
    MW378 : UINT;
    MW379 : UINT;
    MW380 : UINT;
    MW381 : UINT;
    MW382 : UINT;
    MW383 : UINT;
    MW384 : UINT;
    MW385 : UINT;
    MW386 : UINT;
    MW387 : UINT;
    MW388 : UINT;
    MW389 : UINT;
    MW390 : UINT;
    MW391 : UINT;
    MW392 : UINT;
    MW393 : UINT;
    MW394 : UINT;
    MW395 : UINT;
    MW396 : UINT;
    MW397 : UINT;
    MW398 : UINT;
    MW399 : UINT;
    MW400 : UINT;
    MW401 : UINT;
    MW402 : UINT;
    MW403 : UINT;
    MW404 : UINT;
    MW405 : UINT;
    MW406 : UINT;
    MW407 : UINT;
    MW408 : UINT;
    MW409 : UINT;
    MW410 : UINT;
    MW411 : UINT;
    MW412 : UINT;
    MW413 : UINT;
    MW414 : UINT;
    MW415 : UINT;
    MW416 : UINT;
    MW417 : UINT;
    MW418 : UINT;
    MW419 : UINT;
    MW420 : UINT;
    MW421 : UINT;
    MW422 : UINT;
    MW423 : UINT;
    MW424 : UINT;
    MW425 : UINT;
    MW426 : UINT;
    MW427 : UINT;
    MW428 : UINT;
    MW429 : UINT;
    MW430 : UINT;
    MW431 : UINT;
    MW432 : UINT;
    MW433 : UINT;
    MW434 : UINT;
    MW435 : UINT;
    MW436 : UINT;
    MW437 : UINT;
    MW438 : UINT;
    MW439 : UINT;
    MW440 : UINT;
    MW441 : UINT;
    MW442 : UINT;
    MW443 : UINT;
    MW444 : UINT;
    MW445 : UINT;
    MW446 : UINT;
    MW447 : UINT;
    MW448 : UINT;
    MW449 : UINT;
    MW450 : UINT;
    MW451 : UINT;
    MW452 : UINT;
    MW453 : UINT;
    MW454 : UINT;
    MW455 : UINT;
    MW456 : UINT;
    MW457 : UINT;
    MW458 : UINT;
    MW459 : UINT;
    MW460 : UINT;
    MW461 : UINT;
    MW462 : UINT;
    MW463 : UINT;
    MW464 : UINT;
    MW465 : UINT;
    MW466 : UINT;
    MW467 : UINT;
    MW468 : UINT;
    MW469 : UINT;
    MW470 : UINT;
    MW471 : UINT;
    MW472 : UINT;
    MW473 : UINT;
    MW474 : UINT;
    MW475 : UINT;
    MW476 : UINT;
    MW477 : UINT;
    MW478 : UINT;
    MW479 : UINT;
    MW480 : UINT;
    MW481 : UINT;
    MW482 : UINT;
    MW483 : UINT;
    MW484 : UINT;
    MW485 : UINT;
    MW486 : UINT;
    MW487 : UINT;
    MW488 : UINT;
    MW489 : UINT;
    MW490 : UINT;
    MW491 : UINT;
    MW492 : UINT;
    MW493 : UINT;
    MW494 : UINT;
    MW495 : UINT;
    MW496 : UINT;
    MW497 : UINT;
    MW498 : UINT;
    MW499 : UINT;
    MW500 : UINT;
    MW501 : UINT;
    MW502 : UINT;
    MW503 : UINT;
    MW504 : UINT;
    MW505 : UINT;
    MW506 : UINT;
    MW507 : UINT;
    MW508 : UINT;
    MW509 : UINT;
    MW510 : UINT;
    MW511 : UINT;
    MW512 : UINT;
    MW513 : UINT;
    MW514 : UINT;
    MW515 : UINT;
    MW516 : UINT;
    MW517 : UINT;
    MW518 : UINT;
    MW519 : UINT;
    MW520 : UINT;
    MW521 : UINT;
    MW522 : UINT;
    MW523 : UINT;
    MW524 : UINT;
    MW525 : UINT;
    MW526 : UINT;
    MW527 : UINT;
    MW528 : UINT;
    MW529 : UINT;
    MW530 : UINT;
    MW531 : UINT;
    MW532 : UINT;
    MW533 : UINT;
    MW534 : UINT;
    MW535 : UINT;
    MW536 : UINT;
    MW537 : UINT;
    MW538 : UINT;
    MW539 : UINT;
    MW540 : UINT;
    MW541 : UINT;
    MW542 : UINT;
    MW543 : UINT;
    MW544 : UINT;
    MW545 : UINT;
    MW546 : UINT;
    MW547 : UINT;
    MW548 : UINT;
    MW549 : UINT;
    MW550 : UINT;
    MW551 : UINT;
    MW552 : UINT;
    MW553 : UINT;
    MW554 : UINT;
    MW555 : UINT;
    MW556 : UINT;
    MW557 : UINT;
    MW558 : UINT;
    MW559 : UINT;
    MW560 : UINT;
    MW561 : UINT;
    MW562 : UINT;
    MW563 : UINT;
    MW564 : UINT;
    MW565 : UINT;
    MW566 : UINT;
    MW567 : UINT;
    MW568 : UINT;
    MW569 : UINT;
    MW570 : UINT;
    MW571 : UINT;
    MW572 : UINT;
    MW573 : UINT;
    MW574 : UINT;
    MW575 : UINT;
    MW576 : UINT;
    MW577 : UINT;
    MW578 : UINT;
    MW579 : UINT;
    MW580 : UINT;
    MW581 : UINT;
    MW582 : UINT;
    MW583 : UINT;
    MW584 : UINT;
    MW585 : UINT;
    MW586 : UINT;
    MW587 : UINT;
    MW588 : UINT;
    MW589 : UINT;
    MW590 : UINT;
    MW591 : UINT;
    MW592 : UINT;
    MW593 : UINT;
    MW594 : UINT;
    MW595 : UINT;
    MW596 : UINT;
    MW597 : UINT;
    MW598 : UINT;
    MW599 : UINT;
    MW600 : UINT;
    MW601 : UINT;
    MW602 : UINT;
    MW603 : UINT;
    MW604 : UINT;
    MW605 : UINT;
    MW606 : UINT;
    MW607 : UINT;
    MW608 : UINT;
    MW609 : UINT;
    MW610 : UINT;
    MW611 : UINT;
    MW612 : UINT;
    MW613 : UINT;
    MW614 : UINT;
    MW615 : UINT;
    MW616 : UINT;
    MW617 : UINT;
    MW618 : UINT;
    MW619 : UINT;
    MW620 : UINT;
    MW621 : UINT;
    MW622 : UINT;
    MW623 : UINT;
    MW624 : UINT;
    MW625 : UINT;
    MW626 : UINT;
    MW627 : UINT;
    MW628 : UINT;
    MW629 : UINT;
    MW630 : UINT;
    MW631 : UINT;
    MW632 : UINT;
    MW633 : UINT;
    MW634 : UINT;
    MW635 : UINT;
    MW636 : UINT;
    MW637 : UINT;
    MW638 : UINT;
    MW639 : UINT;
    MW640 : UINT;
    MW641 : UINT;
    MW642 : UINT;
    MW643 : UINT;
    MW644 : UINT;
    MW645 : UINT;
    MW646 : UINT;
    MW647 : UINT;
    MW648 : UINT;
    MW649 : UINT;
    MW650 : UINT;
    MW651 : UINT;
    MW652 : UINT;
    MW653 : UINT;
    MW654 : UINT;
    MW655 : UINT;
    MW656 : UINT;
    MW657 : UINT;
    MW658 : UINT;
    MW659 : UINT;
    MW660 : UINT;
    MW661 : UINT;
    MW662 : UINT;
    MW663 : UINT;
    MW664 : UINT;
    MW665 : UINT;
    MW666 : UINT;
    MW667 : UINT;
    MW668 : UINT;
    MW669 : UINT;
    MW670 : UINT;
    MW671 : UINT;
    MW672 : UINT;
    MW673 : UINT;
    MW674 : UINT;
    MW675 : UINT;
    MW676 : UINT;
    MW677 : UINT;
    MW678 : UINT;
    MW679 : UINT;
    MW680 : UINT;
    MW681 : UINT;
    MW682 : UINT;
    MW683 : UINT;
    MW684 : UINT;
    MW685 : UINT;
    MW686 : UINT;
    MW687 : UINT;
    MW688 : UINT;
    MW689 : UINT;
    MW690 : UINT;
    MW691 : UINT;
    MW692 : UINT;
    MW693 : UINT;
    MW694 : UINT;
    MW695 : UINT;
    MW696 : UINT;
    MW697 : UINT;
    MW698 : UINT;
    MW699 : UINT;
    MW700 : UINT;
    MW701 : UINT;
    MW702 : UINT;
    MW703 : UINT;
    MW704 : UINT;
    MW705 : UINT;
    MW706 : UINT;
    MW707 : UINT;
    MW708 : UINT;
    MW709 : UINT;
    MW710 : UINT;
    MW711 : UINT;
    MW712 : UINT;
    MW713 : UINT;
    MW714 : UINT;
    MW715 : UINT;
    MW716 : UINT;
    MW717 : UINT;
    MW718 : UINT;
    MW719 : UINT;
    MW720 : UINT;
    MW721 : UINT;
    MW722 : UINT;
    MW723 : UINT;
    MW724 : UINT;
    MW725 : UINT;
    MW726 : UINT;
    MW727 : UINT;
    MW728 : UINT;
    MW729 : UINT;
    MW730 : UINT;
    MW731 : UINT;
    MW732 : UINT;
    MW733 : UINT;
    MW734 : UINT;
    MW735 : UINT;
    MW736 : UINT;
    MW737 : UINT;
    MW738 : UINT;
    MW739 : UINT;
    MW740 : UINT;
    MW741 : UINT;
    MW742 : UINT;
    MW743 : UINT;
    MW744 : UINT;
    MW745 : UINT;
    MW746 : UINT;
    MW747 : UINT;
    MW748 : UINT;
    MW749 : UINT;
    MW750 : UINT;
    MW751 : UINT;
    MW752 : UINT;
    MW753 : UINT;
    MW754 : UINT;
    MW755 : UINT;
    MW756 : UINT;
    MW757 : UINT;
    MW758 : UINT;
    MW759 : UINT;
    MW760 : UINT;
    MW761 : UINT;
    MW762 : UINT;
    MW763 : UINT;
    MW764 : UINT;
    MW765 : UINT;
    MW766 : UINT;
    MW767 : UINT;
    MW768 : UINT;
    MW769 : UINT;
    MW770 : UINT;
    MW771 : UINT;
    MW772 : UINT;
    MW773 : UINT;
    MW774 : UINT;
    MW775 : UINT;
    MW776 : UINT;
    MW777 : UINT;
    MW778 : UINT;
    MW779 : UINT;
    MW780 : UINT;
    MW781 : UINT;
    MW782 : UINT;
    MW783 : UINT;
    MW784 : UINT;
    MW785 : UINT;
    MW786 : UINT;
    MW787 : UINT;
    MW788 : UINT;
    MW789 : UINT;
    MW790 : UINT;
    MW791 : UINT;
    MW792 : UINT;
    MW793 : UINT;
    MW794 : UINT;
    MW795 : UINT;
    MW796 : UINT;
    MW797 : UINT;
    MW798 : UINT;
    MW799 : UINT;
    MW800 : UINT;
    MW801 : UINT;
    MW802 : UINT;
    MW803 : UINT;
    MW804 : UINT;
    MW805 : UINT;
    MW806 : UINT;
    MW807 : UINT;
    MW808 : UINT;
    MW809 : UINT;
    MW810 : UINT;
    MW811 : UINT;
    MW812 : UINT;
    MW813 : UINT;
    MW814 : UINT;
    MW815 : UINT;
    MW816 : UINT;
    MW817 : UINT;
    MW818 : UINT;
    MW819 : UINT;
    MW820 : UINT;
    MW821 : UINT;
    MW822 : UINT;
    MW823 : UINT;
    MW824 : UINT;
    MW825 : UINT;
    MW826 : UINT;
    MW827 : UINT;
    MW828 : UINT;
    MW829 : UINT;
    MW830 : UINT;
    MW831 : UINT;
    MW832 : UINT;
    MW833 : UINT;
    MW834 : UINT;
    MW835 : UINT;
    MW836 : UINT;
    MW837 : UINT;
    MW838 : UINT;
    MW839 : UINT;
    MW840 : UINT;
    MW841 : UINT;
    MW842 : UINT;
    MW843 : UINT;
    MW844 : UINT;
    MW845 : UINT;
    MW846 : UINT;
    MW847 : UINT;
    MW848 : UINT;
    MW849 : UINT;
    MW850 : UINT;
    MW851 : UINT;
    MW852 : UINT;
    MW853 : UINT;
    MW854 : UINT;
    MW855 : UINT;
    MW856 : UINT;
    MW857 : UINT;
    MW858 : UINT;
    MW859 : UINT;
    MW860 : UINT;
    MW861 : UINT;
    MW862 : UINT;
    MW863 : UINT;
    MW864 : UINT;
    MW865 : UINT;
    MW866 : UINT;
    MW867 : UINT;
    MW868 : UINT;
    MW869 : UINT;
    MW870 : UINT;
    MW871 : UINT;
    MW872 : UINT;
    MW873 : UINT;
    MW874 : UINT;
    MW875 : UINT;
    MW876 : UINT;
    MW877 : UINT;
    MW878 : UINT;
    MW879 : UINT;
    MW880 : UINT;
    MW881 : UINT;
    MW882 : UINT;
    MW883 : UINT;
    MW884 : UINT;
    MW885 : UINT;
    MW886 : UINT;
    MW887 : UINT;
    MW888 : UINT;
    MW889 : UINT;
    MW890 : UINT;
    MW891 : UINT;
    MW892 : UINT;
    MW893 : UINT;
    MW894 : UINT;
    MW895 : UINT;
    MW896 : UINT;
    MW897 : UINT;
    MW898 : UINT;
    MW899 : UINT;
    MW900 : UINT;
    MW901 : UINT;
    MW902 : UINT;
    MW903 : UINT;
    MW904 : UINT;
    MW905 : UINT;
    MW906 : UINT;
    MW907 : UINT;
    MW908 : UINT;
    MW909 : UINT;
    MW910 : UINT;
    MW911 : UINT;
    MW912 : UINT;
    MW913 : UINT;
    MW914 : UINT;
    MW915 : UINT;
    MW916 : UINT;
    MW917 : UINT;
    MW918 : UINT;
    MW919 : UINT;
    MW920 : UINT;
    MW921 : UINT;
    MW922 : UINT;
    MW923 : UINT;
    MW924 : UINT;
    MW925 : UINT;
    MW926 : UINT;
    MW927 : UINT;
    MW928 : UINT;
    MW929 : UINT;
    MW930 : UINT;
    MW931 : UINT;
    MW932 : UINT;
    MW933 : UINT;
    MW934 : UINT;
    MW935 : UINT;
    MW936 : UINT;
    MW937 : UINT;
    MW938 : UINT;
    MW939 : UINT;
    MW940 : UINT;
    MW941 : UINT;
    MW942 : UINT;
    MW943 : UINT;
    MW944 : UINT;
    MW945 : UINT;
    MW946 : UINT;
    MW947 : UINT;
    MW948 : UINT;
    MW949 : UINT;
    MW950 : UINT;
    MW951 : UINT;
    MW952 : UINT;
    MW953 : UINT;
    MW954 : UINT;
    MW955 : UINT;
    MW956 : UINT;
    MW957 : UINT;
    MW958 : UINT;
    MW959 : UINT;
    MW960 : UINT;
    MW961 : UINT;
    MW962 : UINT;
    MW963 : UINT;
    MW964 : UINT;
    MW965 : UINT;
    MW966 : UINT;
    MW967 : UINT;
    MW968 : UINT;
    MW969 : UINT;
    MW970 : UINT;
    MW971 : UINT;
    MW972 : UINT;
    MW973 : UINT;
    MW974 : UINT;
    MW975 : UINT;
    MW976 : UINT;
    MW977 : UINT;
    MW978 : UINT;
    MW979 : UINT;
    MW980 : UINT;
    MW981 : UINT;
    MW982 : UINT;
    MW983 : UINT;
    MW984 : UINT;
    MW985 : UINT;
    MW986 : UINT;
    MW987 : UINT;
    MW988 : UINT;
    MW989 : UINT;
    MW990 : UINT;
    MW991 : UINT;
    MW992 : UINT;
    MW993 : UINT;
    MW994 : UINT;
    MW995 : UINT;
    MW996 : UINT;
    MW997 : UINT;
    MW998 : UINT;
    MW999 : UINT;
  END_VAR
  VAR_INPUT
    I : TPos8 := -1;  (* Индекс определения элемента *)
  END_VAR
  VAR_OUTPUT
    DEF : TDef;
  END_VAR

            CASE i OF
0 : DEF := m_def(MW0,MW1,MW2,MW3,MW4,MW5,MW6,MW7,MW8,MW9);
1 : DEF := m_def(MW10,MW11,MW12,MW13,MW14,MW15,MW16,MW17,MW18,MW19);
2 : DEF := m_def(MW20,MW21,MW22,MW23,MW24,MW25,MW26,MW27,MW28,MW29);
3 : DEF := m_def(MW30,MW31,MW32,MW33,MW34,MW35,MW36,MW37,MW38,MW39);
4 : DEF := m_def(MW40,MW41,MW42,MW43,MW44,MW45,MW46,MW47,MW48,MW49);
5 : DEF := m_def(MW50,MW51,MW52,MW53,MW54,MW55,MW56,MW57,MW58,MW59);
6 : DEF := m_def(MW60,MW61,MW62,MW63,MW64,MW65,MW66,MW67,MW68,MW69);
7 : DEF := m_def(MW70,MW71,MW72,MW73,MW74,MW75,MW76,MW77,MW78,MW79);
8 : DEF := m_def(MW80,MW81,MW82,MW83,MW84,MW85,MW86,MW87,MW88,MW89);
9 : DEF := m_def(MW90,MW91,MW92,MW93,MW94,MW95,MW96,MW97,MW98,MW99);

10 : DEF := m_def(MW100,MW101,MW102,MW103,MW104,MW105,MW106,MW107,MW108,MW109);
11 : DEF := m_def(MW110,MW111,MW112,MW113,MW114,MW115,MW116,MW117,MW118,MW119);
12 : DEF := m_def(MW120,MW121,MW122,MW123,MW124,MW125,MW126,MW127,MW128,MW129);
13 : DEF := m_def(MW130,MW131,MW132,MW133,MW134,MW135,MW136,MW137,MW138,MW139);
14 : DEF := m_def(MW140,MW141,MW142,MW143,MW144,MW145,MW146,MW147,MW148,MW149);
15 : DEF := m_def(MW150,MW151,MW152,MW153,MW154,MW155,MW156,MW157,MW158,MW159);
16 : DEF := m_def(MW160,MW161,MW162,MW163,MW164,MW165,MW166,MW167,MW168,MW169);
17 : DEF := m_def(MW170,MW171,MW172,MW173,MW174,MW175,MW176,MW177,MW178,MW179);
18 : DEF := m_def(MW180,MW181,MW182,MW183,MW184,MW185,MW186,MW187,MW188,MW189);
19 : DEF := m_def(MW190,MW191,MW192,MW193,MW194,MW195,MW196,MW197,MW198,MW199);

20 : DEF := m_def(MW200,MW201,MW202,MW203,MW204,MW205,MW206,MW207,MW208,MW209);
21 : DEF := m_def(MW210,MW211,MW212,MW213,MW214,MW215,MW216,MW217,MW218,MW219);
22 : DEF := m_def(MW220,MW221,MW222,MW223,MW224,MW225,MW226,MW227,MW228,MW229);
23 : DEF := m_def(MW230,MW231,MW232,MW233,MW234,MW235,MW236,MW237,MW238,MW239);
24 : DEF := m_def(MW240,MW241,MW242,MW243,MW244,MW245,MW246,MW247,MW248,MW249);
25 : DEF := m_def(MW250,MW251,MW252,MW253,MW254,MW255,MW256,MW257,MW258,MW259);
26 : DEF := m_def(MW260,MW261,MW262,MW263,MW264,MW265,MW266,MW267,MW268,MW269);
27 : DEF := m_def(MW270,MW271,MW272,MW273,MW274,MW275,MW276,MW277,MW278,MW279);
28 : DEF := m_def(MW280,MW281,MW282,MW283,MW284,MW285,MW286,MW287,MW288,MW289);
29 : DEF := m_def(MW290,MW291,MW292,MW293,MW294,MW295,MW296,MW297,MW298,MW299);

30 : DEF := m_def(MW300,MW301,MW302,MW303,MW304,MW305,MW306,MW307,MW308,MW309);
31 : DEF := m_def(MW310,MW311,MW312,MW313,MW314,MW315,MW316,MW317,MW318,MW319);
32 : DEF := m_def(MW320,MW321,MW322,MW323,MW324,MW325,MW326,MW327,MW328,MW329);
33 : DEF := m_def(MW330,MW331,MW332,MW333,MW334,MW335,MW336,MW337,MW338,MW339);
34 : DEF := m_def(MW340,MW341,MW342,MW343,MW344,MW345,MW346,MW347,MW348,MW349);
35 : DEF := m_def(MW350,MW351,MW352,MW353,MW354,MW355,MW356,MW357,MW358,MW359);
36 : DEF := m_def(MW360,MW361,MW362,MW363,MW364,MW365,MW366,MW367,MW368,MW369);
37 : DEF := m_def(MW370,MW371,MW372,MW373,MW374,MW375,MW376,MW377,MW378,MW379);
38 : DEF := m_def(MW380,MW381,MW382,MW383,MW384,MW385,MW386,MW387,MW388,MW389);
39 : DEF := m_def(MW390,MW391,MW392,MW393,MW394,MW395,MW396,MW397,MW398,MW399);

40 : DEF := m_def(MW400,MW401,MW402,MW403,MW404,MW405,MW406,MW407,MW408,MW409);
41 : DEF := m_def(MW410,MW411,MW412,MW413,MW414,MW415,MW416,MW417,MW418,MW419);
42 : DEF := m_def(MW420,MW421,MW422,MW423,MW424,MW425,MW426,MW427,MW428,MW429);
43 : DEF := m_def(MW430,MW431,MW432,MW433,MW434,MW435,MW436,MW437,MW438,MW439);
44 : DEF := m_def(MW440,MW441,MW442,MW443,MW444,MW445,MW446,MW447,MW448,MW449);
45 : DEF := m_def(MW450,MW451,MW452,MW453,MW454,MW455,MW456,MW457,MW458,MW459);
46 : DEF := m_def(MW460,MW461,MW462,MW463,MW464,MW465,MW466,MW467,MW468,MW469);
47 : DEF := m_def(MW470,MW471,MW472,MW473,MW474,MW475,MW476,MW477,MW478,MW479);
48 : DEF := m_def(MW480,MW481,MW482,MW483,MW484,MW485,MW486,MW487,MW488,MW489);
49 : DEF := m_def(MW490,MW491,MW492,MW493,MW494,MW495,MW496,MW497,MW498,MW499);

50 : DEF := m_def(MW500,MW501,MW502,MW503,MW504,MW505,MW506,MW507,MW508,MW509);
51 : DEF := m_def(MW510,MW511,MW512,MW513,MW514,MW515,MW516,MW517,MW518,MW519);
52 : DEF := m_def(MW520,MW521,MW522,MW523,MW524,MW525,MW526,MW527,MW528,MW529);
53 : DEF := m_def(MW530,MW531,MW532,MW533,MW534,MW535,MW536,MW537,MW538,MW539);
54 : DEF := m_def(MW540,MW541,MW542,MW543,MW544,MW545,MW546,MW547,MW548,MW549);
55 : DEF := m_def(MW550,MW551,MW552,MW553,MW554,MW555,MW556,MW557,MW558,MW559);
56 : DEF := m_def(MW560,MW561,MW562,MW563,MW564,MW565,MW566,MW567,MW568,MW569);
57 : DEF := m_def(MW570,MW571,MW572,MW573,MW574,MW575,MW576,MW577,MW578,MW579);
58 : DEF := m_def(MW580,MW581,MW582,MW583,MW584,MW585,MW586,MW587,MW588,MW589);
59 : DEF := m_def(MW590,MW591,MW592,MW593,MW594,MW595,MW596,MW597,MW598,MW599);

60 : DEF := m_def(MW600,MW601,MW602,MW603,MW604,MW605,MW606,MW607,MW608,MW609);
61 : DEF := m_def(MW610,MW611,MW612,MW613,MW614,MW615,MW616,MW617,MW618,MW619);
62 : DEF := m_def(MW620,MW621,MW622,MW623,MW624,MW625,MW626,MW627,MW628,MW629);
63 : DEF := m_def(MW630,MW631,MW632,MW633,MW634,MW635,MW636,MW637,MW638,MW639);
64 : DEF := m_def(MW640,MW641,MW642,MW643,MW644,MW645,MW646,MW647,MW648,MW649);
65 : DEF := m_def(MW650,MW651,MW652,MW653,MW654,MW655,MW656,MW657,MW658,MW659);
66 : DEF := m_def(MW660,MW661,MW662,MW663,MW664,MW665,MW666,MW667,MW668,MW669);
67 : DEF := m_def(MW670,MW671,MW672,MW673,MW674,MW675,MW676,MW677,MW678,MW679);
68 : DEF := m_def(MW680,MW681,MW682,MW683,MW684,MW685,MW686,MW687,MW688,MW689);
69 : DEF := m_def(MW690,MW691,MW692,MW693,MW694,MW695,MW696,MW697,MW698,MW699);

70 : DEF := m_def(MW700,MW701,MW702,MW703,MW704,MW705,MW706,MW707,MW708,MW709);
71 : DEF := m_def(MW710,MW711,MW712,MW713,MW714,MW715,MW716,MW717,MW718,MW719);
72 : DEF := m_def(MW720,MW721,MW722,MW723,MW724,MW725,MW726,MW727,MW728,MW729);
73 : DEF := m_def(MW730,MW731,MW732,MW733,MW734,MW735,MW736,MW737,MW738,MW739);
74 : DEF := m_def(MW740,MW741,MW742,MW743,MW744,MW745,MW746,MW747,MW748,MW749);
75 : DEF := m_def(MW750,MW751,MW752,MW753,MW754,MW755,MW756,MW757,MW758,MW759);
76 : DEF := m_def(MW760,MW761,MW762,MW763,MW764,MW765,MW766,MW767,MW768,MW769);
77 : DEF := m_def(MW770,MW771,MW772,MW773,MW774,MW775,MW776,MW777,MW778,MW779);
78 : DEF := m_def(MW780,MW781,MW782,MW783,MW784,MW785,MW786,MW787,MW788,MW789);
79 : DEF := m_def(MW790,MW791,MW792,MW793,MW794,MW795,MW796,MW797,MW798,MW799);

80 : DEF := m_def(MW800,MW801,MW802,MW803,MW804,MW805,MW806,MW807,MW808,MW809);
81 : DEF := m_def(MW810,MW811,MW812,MW813,MW814,MW815,MW816,MW817,MW818,MW819);
82 : DEF := m_def(MW820,MW821,MW822,MW823,MW824,MW825,MW826,MW827,MW828,MW829);
83 : DEF := m_def(MW830,MW831,MW832,MW833,MW834,MW835,MW836,MW837,MW838,MW839);
84 : DEF := m_def(MW840,MW841,MW842,MW843,MW844,MW845,MW846,MW847,MW848,MW849);
85 : DEF := m_def(MW850,MW851,MW852,MW853,MW854,MW855,MW856,MW857,MW858,MW859);
86 : DEF := m_def(MW860,MW861,MW862,MW863,MW864,MW865,MW866,MW867,MW868,MW869);
87 : DEF := m_def(MW870,MW871,MW872,MW873,MW874,MW875,MW876,MW877,MW878,MW879);
88 : DEF := m_def(MW880,MW881,MW882,MW883,MW884,MW885,MW886,MW887,MW888,MW889);
89 : DEF := m_def(MW890,MW891,MW892,MW893,MW894,MW895,MW896,MW897,MW898,MW899);

90 : DEF := m_def(MW900,MW901,MW902,MW903,MW904,MW905,MW906,MW907,MW908,MW909);
91 : DEF := m_def(MW910,MW911,MW912,MW913,MW914,MW915,MW916,MW917,MW918,MW919);
92 : DEF := m_def(MW920,MW921,MW922,MW923,MW924,MW925,MW926,MW927,MW928,MW929);
93 : DEF := m_def(MW930,MW931,MW932,MW933,MW934,MW935,MW936,MW937,MW938,MW939);
94 : DEF := m_def(MW940,MW941,MW942,MW943,MW944,MW945,MW946,MW947,MW948,MW949);
95 : DEF := m_def(MW950,MW951,MW952,MW953,MW954,MW955,MW956,MW957,MW958,MW959);
96 : DEF := m_def(MW960,MW961,MW962,MW963,MW964,MW965,MW966,MW967,MW968,MW969);
97 : DEF := m_def(MW970,MW971,MW972,MW973,MW974,MW975,MW976,MW977,MW978,MW979);
98 : DEF := m_def(MW980,MW981,MW982,MW983,MW984,MW985,MW986,MW987,MW988,MW989);
99 : DEF := m_def(MW990,MW991,MW992,MW993,MW994,MW995,MW996,MW997,MW998,MW999);
END_CASE;
          
END_FUNCTION_BLOCK

(* Чтение элемента из регистров *)
FUNCTION_BLOCK ReadItem
  VAR_EXTERNAL
    HDR : THead;  (* Внешний заголовок модели *)
  END_VAR
  VAR_INPUT
    PIT : TPos8 := -1;  (* Индекс элемента *)
  END_VAR
  VAR_OUTPUT
    iRes : TError := E_SUCCESS;  (* Результат блока *)
  END_VAR
  VAR
    Def : TDef;  (* Определение элемента *)
    Item : TItem;  (* Элемент (локальная копия) *)
    Shape : TShape;  (* Геометрия (локальная копия) *)
    Off : P_INT;  (* Смещение в сетке *)
    msg : STRING;  (* Строка в протокол *)
    _GetDef : GetDef;  (* Чтение заголовка из регистров *)
  END_VAR

            iRes:=E_SUCCESS;

(* Проверка корректности индекса элемента *)
if (PIT < 0 or PIT >= HDR.Ni) then iRes:=E_INDEX; {goto __exit} end_if;

(* Получение определения элемента из массива конфигурации *)
_GetDef(i := PIT, DEF => Def);

(* Проверка индексов в массивах VAL, MAT, KNT *)
if (HDR.Nv<>0 and Def.Iv >= HDR.Nv) then iRes:=E_VALUE; {goto __exit} end_if;
if (HDR.Nm=0  or  Def.Im >= HDR.Nm) then iRes:=E_MATER; {goto __exit} end_if;
if (HDR.Ng=0  or  Def.Ig >= HDR.Ng) then iRes:=E_GRID;  {goto __exit} end_if;

(* Инициализация *)
Item.ID  := Def.ID;  (* Копирование идентификатора элемента          *)
Item.Im  := Def.Im;  (* Копирование индекса материала                *)
Item.Iv  := Def.Iv;  (* Копирование индекса величины (если есть)     *)
Item.Par := -1;      (* Родитель не определен, дерево строится позже *)
Item.Num := 0;       (* Детей пока тоже нет, дерево строится позже   *)

(* Флаги геометрии (расшифровка в Do_Validate)  *)
Shape.wF  := Def.CF;   

(* Временное размещение начальных смещений в Кn (int[0..2]) *)
Shape.Kn[0] := Def.R0;                       (* начальный радиус (X0) *)
Shape.Kn[1] := 
  WORD_TO_INT(SHR((Def.CF and 16#0F00), 8)); (* начальный сектор (Y0) *)
Shape.Kn[2] := 0;                            (* начальная высота (Z0) *)

(* Копирование xyz[], lwh[] *)
Shape.pL[0] := INT_TO_REAL(Def.XYZ[0]);
Shape.pL[1] := INT_TO_REAL(Def.XYZ[1]);
Shape.pL[2] := INT_TO_REAL(Def.XYZ[2]);
Shape.Lx[0] := INT_TO_REAL(Def.LWH[0]);
Shape.Lx[1] := INT_TO_REAL(Def.LWH[1]);
Shape.Lx[2] := INT_TO_REAL(Def.LWH[2]);

(* Завершение процедуры *)
{__exit:}
if (iRes = E_SUCCESS) then 
  PIT := set_sh(PIT, Shape);
  PIT := set_it(PIT, Item);
end_if;

          
END_FUNCTION_BLOCK

(* Проверка корректности модели *)
FUNCTION Do_Validate : BOOL
  VAR_INPUT
    PIT : TPos8 := -1;  (* Первичный узел проверки *)
  END_VAR
  VAR
    It : TIter;  (* Итератор *)
    Item : TItem;  (* Элемент *)
    Sh : TShape;  (* Геометрия элемента *)
    Ax : USINT := 0;  (* Флаг "ось задана" *)
    bAx : BOOL := false;  (* Флаг "ось задана" *)
    bCx : BOOL := false;  (* Флаг "цилиндрическая система" *)
    bOx : BOOL := false;  (* Флаг "задана точка отсчёта" *)
    OFF : P_INT;  (* Cмещение и размер ячейки GRid по индексам *)
    i : INT := 0;  (* Индекс цикла 1 *)
    j : INT := 0;  (* Индекс цикла 2 *)
    k : INT := 0;  (* Индекс цикла 3 *)
    m : INT := 0;  (* Индекс цикла 4 *)
    iP : TPos8 := 0;  (* Индекс родителя *)
    P0 : TPoint := [0.0, 0.0, 0.0];  (* Точка начала отсчёта *)
    Lx : TPoint := [0.0, 0.0, 0.0];  (* Линейные габариты *)
    O : TAxO;  (* Индексы координат x, y, z *)
    RI : ARRAY[0..2] OF P_RESI;  (* Массив упорядоченных пар (значение-индекс) *)
    temp : P_RESI;  (* Ячейка для перестановки при сортировке *)
    rTemp : REAL := 0.0;  (* Начальная температура ячейки *)
    bRes : BOOL := false;  (* флаг результата *)
  END_VAR
  VAR CONSTANT
    PI : REAL := 180.0;  (* Число Пи *)
    PI2 : REAL := 360.0;  (* Число 2*Пи *)
    PI_RAD : REAL := 3.1415926535897932384626433832795;  (* Число 2*Пи (радиан) *)
  END_VAR

            Do_Validate := st_check(false);
if (not Do_Validate) then return; end_if;

(* Обход дерева элементов *)
it := it_begin(ID2PIT(0));
while (it.item<>-1) do
  (* Локальная копия элемента *)
  Item  := get_it(it.item);
  Sh    := get_sh(it.item);
  
  (* Расшифровка гео-флагов *)
  (* Флаги границ  - 0-7 биты в wF *)
  (* Sh.bF := WORD_TO_BYTE(Sh.wF AND 16#00FF); *)
  
  (* Номер сектора скопирован в Sh.Kn[1] в ReadItem() *)
  (*Item.nS := WORD_TO_USINT(SHR((Def.CF AND 16#0F00), 8)); *)

  (* Флаг составного элемента - 16 бит (не используется) *)
  (* Item.bP := ((Def.CF AND 16#8000)<>0); *)
  
  (* Ось симметрии - следующие 12-13 биты в wF *)
  Ax  := WORD_TO_USINT(SHR((Sh.wF AND 16#3000), 12));

  bCx := ((Sh.wF and 16#4000)<>0); (* Признак 'цилиндрич. система'   *)
  bAx := (Ax<>0);                  (* Признак 'ось задана'           *)
  bOx := (not bCx or bAx);         (* Признак 'задана точка отсчёта' *)

  case (it.dir) of
  DIR_DOWN:
    (* Определение точек начала отсчёта (НО) в ABS координатах   *)
    if (Item.Num>0 and bOx) then   (* Элемент с новой точкой отсчёта *)
      (* Прибавляем координаты НО к накопителю P0 *)
      P0[0] := P0[0] + Sh.pL[0]; 
      P0[1] := P0[1] + Sh.pL[1]; 
      P0[2] := P0[2] + Sh.pL[2];
    end_if;
    
  DIR_UP:
    (* Определение точек начала отсчёта в ABS координатах *)
    if (Item.Num>0 and bOx) then  (* Элемент с новой точкой отсчёта *)
      (* Вычитаем координаты НО из накопителя P0 *)
      P0[0] := P0[0] - Sh.pL[0]; 
      P0[1] := P0[1] - Sh.pL[1]; 
      P0[2] := P0[2] - Sh.pL[2];
    end_if;
    
    (* Сохраняем собственную точку НО *)
    Sh.p0[0] := P0[0]; 
    Sh.p0[1] := P0[1];
    Sh.p0[2] := P0[2];
    
    (* === Цилиндрическая система === *)
    if (bCx) then
    
      (* Если ось не задана - она наследуется от родителя *)
      if (not bAx)  then
        iP := Item.Par;
        while (iP<>-1) do
          Ax := sh_get_ax(get_sh(iP));
          iP := it_ip(iP);
          if (Ax<>0) then exit; end_if;
        end_while;
        if (Ax=0) then {goto __error} end_if;
      end_if;

      (* Индексы "оригинальных" координат: Ax -> O *)
       O := AxO(Ax);
       
      (* --- Преобразование начальной точки --- *)
      if (bAx) then
        (* Если ось задана:       *)
        (* (1) XYZ->OOO (декарт); *)
        Sh.p0[0]   := Sh.p0[0] + Sh.pL[0];
        Sh.p0[1]   := Sh.p0[1] + Sh.pL[1];
        Sh.p0[2]   := Sh.p0[2] + Sh.pL[2];
        
        (* (2) R0->X, nS->Y, Z=0  *)
        Sh.pL[O.x] := INT_TO_REAL(Sh.Kn[0]);            (* R0  *)
        Sh.pL[O.y] := INT_TO_REAL(Sh.Kn[1]) *(PI/8.0);  (* nS  *)
        Sh.pL[O.z] := INT_TO_REAL(Sh.Kn[2]);            (* 0.0 *)
      end_if;
      
      (* Приведение угловой координаты к диапазону [-PI..PI] *)
      Sh.pL[O.y]:=angle(Sh.pL[O.y], (-PI));
      
      (* Приведение углового размера   к диапазону [0..2*PI] *)
      Sh.Lx[O.y]:=angle(Sh.Lx[O.y], 0.0);
      
      (* Если размер =0 -> делаем его =360град *)
      if (Sh.Lx[O.y]=0.0) then Sh.Lx[O.y]:=PI2; end_if;
      
    else  (* Прямоугольные координаты *)
      Ax := 0;
    end_if;
    
    (* Установка флагов оси симметрии Ax *)
    Sh := sh_set_ax(Sh, Ax);
    
    (* === Расчёт сетки BEGIN === *)
    Lx:=Sh.Lx;
    
    (* Вычисление радиального размера *)
    if (Ax<>0) then Lx[O.y]:=Lx[O.x]*Lx[O.y]*PI_RAD/360.0; end_if;
    
    (* Инициализация перед сортировкой пар 'размер-индекс' *) 
    RI[0].A := Lx[0]; RI[0].B := 0;
    RI[1].A := Lx[1]; RI[1].B := 1;
    RI[2].A := Lx[2]; RI[2].B := 2;
    
    (* Сортировка пузырьком пар 'размер-индекс' *) 
    for i:=0 to 1 do
      for  j:=0 to 1-i do
        if (RI[j].A > RI[j+1].A) then
          temp:=RI[j]; RI[j]:=RI[j+1]; RI[j+1]:=temp;
        end_if;
      end_for;
    end_for;
    
    (* Определяем количество узлов сети (Kn) *)
    if ((RI[1].A+RI[2].A)/RI[0].A > 4.0) then
      Sh.Kn[RI[0].B]:=8;
      if ((RI[2].A/RI[1].A) > 4.0) then
        Sh.Kn[RI[1].B]:=8;  
        Sh.Kn[RI[2].B]:=64;
      else
        Sh.Kn[RI[1].B]:=16; 
        Sh.Kn[RI[2].B]:=32;
      end_if;
    else
      Sh.Kn[0]:=16; 
      Sh.Kn[1]:=16; 
      Sh.Kn[2]:=16;
    end_if;
    (* === Расчёт сетки END === *)

  end_case;

  (* TEST -> *)
  if not (
    (it.item>=1 and it.item<=99) 
  ) then 
    Item.Im := 0; (* воздух *)
  end_if;
  (* <- TEST *)

  (* Записываем "валидный" элемент ОБРАТНО в массив *)
  it.item := set_sh(it.item, Sh);
  it.item := set_it(it.item, Item);
  
  (* === Инициализация сетки элемента === *)
  it.item := IT_InitTemp(it.item, 20.0, true);
  
  it := it_next(it);
end_while;

(*PIT := IT_InitTemp(42, 100.0, true);*)

Do_Validate := true;
return;

{ __error: }
Do_Validate := false;

          
END_FUNCTION

(* Проверка корректности модели *)
FUNCTION Do_CheckValid : BOOL
  VAR_INPUT
    PIT : TPos8 := -1;  (* Первичный узел проверки *)
  END_VAR
  VAR
    PIT2 : TPos8 := 0;  (* Вторичный узел проверки *)
    bRes : BOOL := false;  (* Флаг результата *)
    It : TIter;  (* Итератор *)
    stack : ARRAY[0..99] OF TPos8;  (* Стек элементов *)
    kids : ARRAY[0..15] OF TPos8;  (* Выборка потомства из стека *)
    n : SINT := 0;  (* Количество элементов в стеке *)
    m : SINT := 0;  (* Количество детей в выборке *)
    im : SINT := 0;  (* Индекс цикла 1 *)
    j : SINT := 0;  (* Индекс цикла 2 *)
    Chk : TDot;  (* Результат проверки точки *)
    bC : BOOL := false;  (* Флаг 'элемент в цилиндрической СК' *)
    Sh : TShape;  (* Фигура элемента *)
    p0 : TPoint;  (* Точка 0 элемента *)
    p1 : TPoint;  (* Точка 1 элемента *)
    p2 : TPoint;  (* Точка 2 элемента *)
    msg : STRING := '';  (* Строка состояния *)
  END_VAR

            Do_CheckValid := st_check(false);
if (not Do_CheckValid) then return; end_if;

(* Обход дерева элементов *)
it := it_begin(ID2PIT(0));
while (it.item<>-1) do

